REGION Network 80: Check for Parameter Format Type
   RUNG wire#powerrail
      Contact( #ALLWAYS_ON )
      { S7_GenerateENO := "TRUE" } Move(in := #PARA_INTERNAL_DPV1.Responce.Format, out1 => #Response_Format_Dummy)
      wire#w1
      { S7_Templates := "SrcType := Int" } EQ_Contact(in1 := #Response_Format_Dummy, in2 := 67)
      wire#w2
      Coil( #Format_Check_1 )
   END_RUNG
   RUNG wire#w1
      { S7_Templates := "SrcType := Int" } EQ_Contact(in1 := #Response_Format_Dummy, in2 := 4)
   END_RUNG wire#w2
   RUNG wire#w1
      { S7_Templates := "SrcType := Int" } EQ_Contact(in1 := #Response_Format_Dummy, in2 := 7)
   END_RUNG wire#w2
   // the same network as SCL:
   // ENO of a box is taken as its EN; it also drops when the box reports an error
   IF #ALLWAYS_ON THEN #Response_Format_Dummy := #PARA_INTERNAL_DPV1.Responce.Format; END_IF;
   #Format_Check_1 := #ALLWAYS_ON AND ((#Response_Format_Dummy = 67) OR (#Response_Format_Dummy = 4) OR (#Response_Format_Dummy = 7));
END_REGION

REGION Network 81: Wrtie parameter area DP-V1
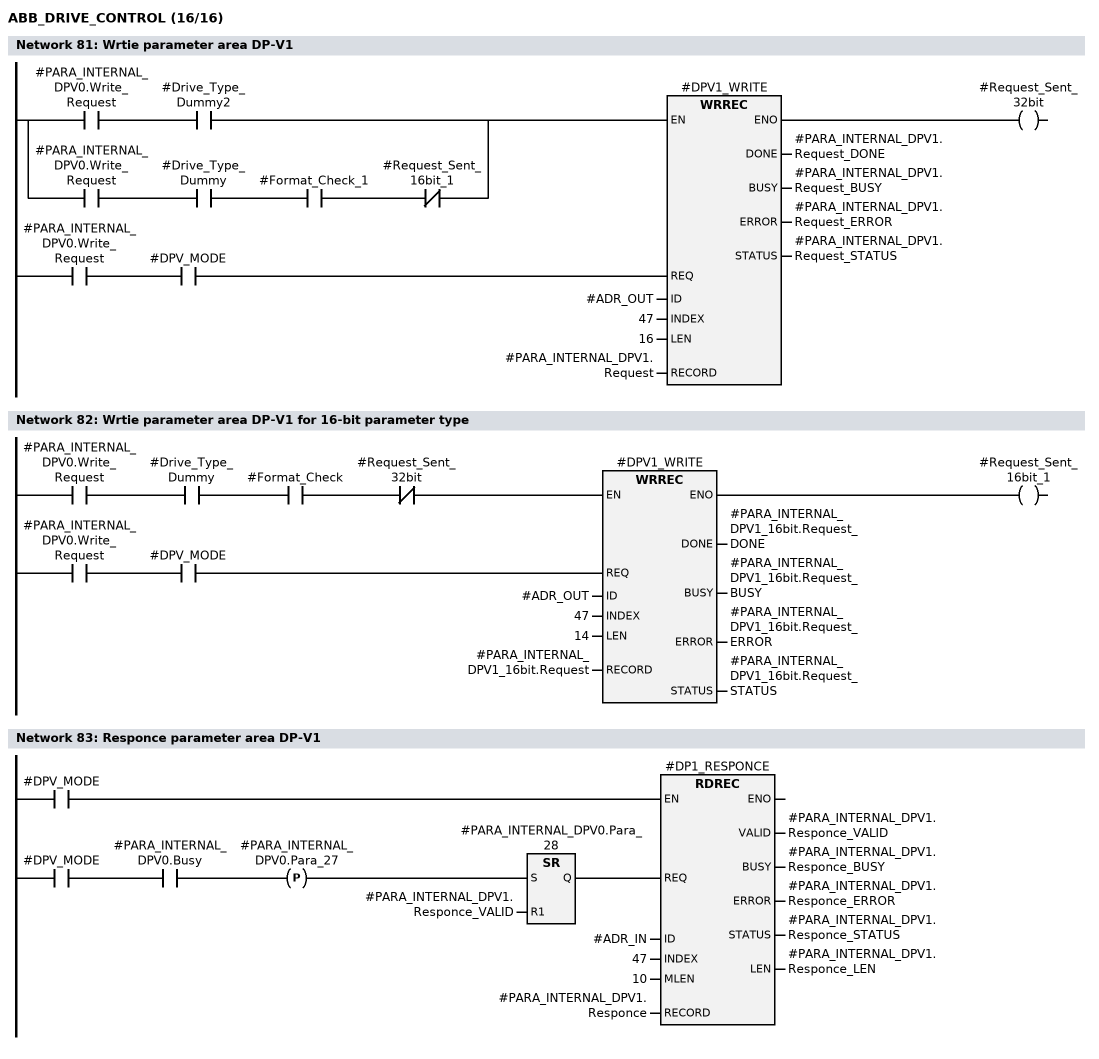
   // ENO of a box is taken as its EN; it also drops when the box reports an error
   #_w1 := (#PARA_INTERNAL_DPV0.Write_Request AND #Drive_Type_Dummy2) OR (#PARA_INTERNAL_DPV0.Write_Request AND #Drive_Type_Dummy AND #Format_Check_1 AND NOT #Request_Sent_16bit_1);
   IF #_w1 THEN
       #DPV1_WRITE(REQ := #PARA_INTERNAL_DPV0.Write_Request AND #DPV_MODE,   // WRREC
                   ID := #ADR_OUT,
                   INDEX := 47,
                   LEN := 16,
                   RECORD := #PARA_INTERNAL_DPV1.Request,
                   DONE => #PARA_INTERNAL_DPV1.Request_DONE,
                   BUSY => #PARA_INTERNAL_DPV1.Request_BUSY,
                   ERROR => #PARA_INTERNAL_DPV1.Request_ERROR,
                   STATUS => #PARA_INTERNAL_DPV1.Request_STATUS);
   END_IF;
   #Request_Sent_32bit := #_w1;
END_REGION

REGION Network 82: Wrtie parameter area DP-V1 for 16-bit parameter type
   // ENO of a box is taken as its EN; it also drops when the box reports an error
   #_w1 := #PARA_INTERNAL_DPV0.Write_Request AND #Drive_Type_Dummy AND #Format_Check AND NOT #Request_Sent_32bit;
   IF #_w1 THEN
       #DPV1_WRITE(REQ := #PARA_INTERNAL_DPV0.Write_Request AND #DPV_MODE,   // WRREC
                   ID := #ADR_OUT,
                   INDEX := 47,
                   LEN := 14,
                   RECORD := #PARA_INTERNAL_DPV1_16bit.Request,
                   DONE => #PARA_INTERNAL_DPV1_16bit.Request_DONE,
                   BUSY => #PARA_INTERNAL_DPV1_16bit.Request_BUSY,
                   ERROR => #PARA_INTERNAL_DPV1_16bit.Request_ERROR,
                   STATUS => #PARA_INTERNAL_DPV1_16bit.Request_STATUS);
   END_IF;
   #Request_Sent_16bit_1 := #_w1;
END_REGION

REGION Network 83: Responce parameter area DP-V1
   #_w1 := #DPV_MODE AND #PARA_INTERNAL_DPV0.Busy;
   #_w2 := #_w1 AND NOT #PARA_INTERNAL_DPV0.Para_27;   // rising edge
   #PARA_INTERNAL_DPV0.Para_27 := #_w1;
   IF #_w2 THEN
       #PARA_INTERNAL_DPV0.Para_28 := TRUE;   // SR flip-flop
   END_IF;
   IF #PARA_INTERNAL_DPV1.Responce_VALID THEN #PARA_INTERNAL_DPV0.Para_28 := FALSE; END_IF;
   IF #DPV_MODE THEN
       #DP1_RESPONCE(REQ := #PARA_INTERNAL_DPV0.Para_28,   // RDREC
                     ID := #ADR_IN,
                     INDEX := 47,
                     MLEN := 10,
                     RECORD := #PARA_INTERNAL_DPV1.Responce,
                     VALID => #PARA_INTERNAL_DPV1.Responce_VALID,
                     BUSY => #PARA_INTERNAL_DPV1.Responce_BUSY,
                     ERROR => #PARA_INTERNAL_DPV1.Responce_ERROR,
                     STATUS => #PARA_INTERNAL_DPV1.Responce_STATUS,
                     LEN => #PARA_INTERNAL_DPV1.Responce_LEN);
   END_IF;
END_REGION
END_FUNCTION_BLOCK

FUNCTION_BLOCK "ACS_DRIVE_PARA"   // FB501, LAD
TITLE = ACS_DRIVE_PARA
{ S7_Optimized_Access := 'FALSE' }
AUTHOR : ABB
FAMILY : DRIVES
NAME : ABB
VERSION : 1.2
   VAR_INPUT
      ADR_IN : Hw_Io;   // 1: Address of first input byte
      ADR_OUT : Hw_Io;   // 2: Address of first output byte
      READ : Bool;   // 3: Read parameter value
      WRITE : Bool;   // 4: Write parameter value
      PARAM_NUM : DInt;   // 5: Parameter number: 3 digits = group, 2 digits = index; e.g Par 20.06 = 2006
      VALUE_IN : DInt;   // 6: Write parameter value
      DRIVE : DB_ANY;   // 8: Instance of the ABB_DRIVE_CONTROL_FB
      THIS_BLOCK_DB : DB_ANY;
   END_VAR
   VAR_OUTPUT
      DONE : Bool;   // 1: Pulse execution finished
      ERR : Bool;   // 2: Error occured
      ERNO : Word;   // 3: Error ID
      BUSY : Bool;   // 4: Function block busy
      PARAM_NUM_OUT : DInt;   // 5: Parameter number: 3 digits = group, 2 digits = index; e.g Par 20.06 = 2006
      VALUE_OUT : DInt;   // 6: Readed parameter value
   END_VAR
   VAR
      PARA_INTERNAL : Struct
         Done : Bool;
         Err : Bool;
         Busy : Bool;
         Read_FB : Bool;
         Write_FB : Bool;
         Time_out : Bool;
         Read_request : Bool;
         Write_Request : Bool;
         Parameter_access : Bool;
         para_err : Bool;
         Para_10 : Bool;
         DPV1_DONE : Bool;
         Para_12 : Bool;
         Para_13 : Bool;
         Para_14 : Bool;
         Para_15 : Bool;
         Para_16 : Bool;
         Para_17 : Bool;
         Para_18 : Bool;
         Para_19 : Bool;
         Para_20 : Bool;
         Para_21 : Bool;
         Para_22 : Bool;
         Para_23 : Bool;
         Para_24 : Bool;
         Para_25 : Bool;
         Para_26 : Bool;
         Para_27 : Bool;
         Para_28 : Bool;
         Para_29 : Bool;
         Para_30 : Bool;
         DPV_MODE : Bool;   // DP-V0 = 0 (false) / DP-V1 = 1 (true)
         RESPONCE_LABEL : Int;
         PARA_NUM_OUT : Int;
         PARA_NUM_INDEX_OUT : Int;
         PARA_ERR_NRO : Word;
         PARA_VALUE_OUT : DInt;
         ADDRESS_IN : Word;
         ADDRESS_OUT : Word;
         Master_to_Slave : Struct
            ID : Word;   // Request Label bits 4-7 Parameter number bits 0-2
            IND : Word;   // Parameter number index bits 0-15
            VALUE : DWord;   // Parameter values
         END_STRUCT;
         Slave_to_Master : Struct
            ID : Word;   // Request Label bits 4-7 Parameter number bits 0-2
            IND : Word;   // Parameter number index bits 0-15
            VALUE : DWord;   // Parameter values
         END_STRUCT;
         PPO_TYPE : Int;   // PPO-Type: 1,2,3,4,5 or 6; 0 = no function
         ADAPTER_TYPE : Int;   // AdapterType:FPBA=1,RPBA=2,FENA=3
         DRIVE_TYPE : Int;   // ACS800=1,ACSM1=2,ACS350=3,ACS355=4,ACS550=5,ACS850=6,ACS880=7,ACS580=8,ACS380=9
      END_STRUCT;
      ReadCommand : Int;
      WriteCommand : Int;
      PARA_NUM_IN : Int;
      PARA_NUM_ON_RPBA : Bool;
      PARA_NUM_ON_FPBA : Bool;
      PARANUM_DINT : DInt;
      PARA_ERR : Bool;
      ITERNAL_READ_ERR : Int;
      ITERNAL_ERITE_ERR : Int;
      TEMP_PARA_NUM : DInt;
      Allways_ON : Bool;
      Allways_OFF : Bool;
      Dummy : Bool;
      TEMPPI : DInt;
      START_VALUE : DInt;
      ZERO_VALUE : DInt;
      PARA_INTERNAL_DPV1 : Struct
         Request : Struct
            Reference : Byte;
            ID : Byte;
            Axis : Byte;
            NoOfParameters : Byte;
            Attribute : Byte;
            NoOfElements : Byte;
            ParameterIndex : Word;
            Subindex : Word;
            Format : Byte;
            NumberOfValues : Byte;
            Value : DWord;
         END_STRUCT;
         Responce : Struct
            Reference : Byte;
            ID : Byte;
            Axis : Byte;
            NoOfParametrs : Byte;
            Format : Byte;
            NoOfValues : Byte;
            Value : DWord;
         END_STRUCT;
         Request_DONE : Bool;
         Request_BUSY : Bool;
         Request_ERROR : Bool;
         Request_STATUS : DWord;
         Responce_VALID : Bool;
         Responce_BUSY : Bool;
         Responce_ERROR : Bool;
         Responce_STATUS : DWord;
         Responce_LEN : UInt;
      END_STRUCT;
      Drive_Dummy1 : Bool;
      Drive_Dummy2 : Bool;
      PARA_INTERNAL_DPV1_16bit : Struct
         Request : Struct
            Reference : Byte;
            ID : Byte;
            Axis : Byte;
            NoOfParameters : Byte;
            Attribute : Byte;
            NoOfElements : Byte;
            ParameterIndex : Word;
            Subindex : Word;
            Format : Byte;
            NumberOfValues : Byte;
            Value : Word;
         END_STRUCT;
         Responce : Struct
            Reference : Byte;
            ID : Byte;
            Axis : Byte;
            NoOfParametrs : Byte;
            Format : Byte;
            NoOfValues : Byte;
            Value : DWord;
         END_STRUCT;
         Request_DONE : Bool;
         Request_BUSY : Bool;
         Request_ERROR : Bool;
         Request_STATUS : DWord;
         Responce_VALID : Bool;
         Responce_BUSY : Bool;
         Responce_ERROR : Bool;
         Responce_STATUS : DWord;
         Responce_LEN : Int;
      END_STRUCT;
      PARA32bit_Read : Bool;
      PARA16bit_Read : Bool;
   END_VAR
   VAR_TEMP
      PARAM_NUM_Temp : Int;
      ReadCommand_Temp : Int;
      PARAM_NUM_Temp2 : Int;
      WriteCommand_Temp : Int;
      PARA_INTERNAL_Slave_to_Master_ID_Temp : Word;
      PARA_INTERNAL_Slave_to_Master_ID_Temp2 : Word;
      PARA_INTERNAL_Slave_to_Master_ID_Temp3 : Word;
      PARA_INTERNAL_Slave_to_Master_IND_Temp : Word;
      PARA_INTERNAL_Master_to_Slave_ID_Temp : DInt;
      PARA_INTERNAL_Master_to_Slave_ID_Num_Temp : DInt;
      PARA_INTERNAL_Master_to_Slave_ID_Num_Temp2 : Int;
      ReadCommand_Temp2 : Word;
      PARA_INTERNAL_Master_to_Slave_ID_Temp2 : DInt;
      PARA_INTERNAL_Master_to_Slave_ID_Num_Temp3 : DInt;
      PARA_INTERNAL_Master_to_Slave_ID_Num_Temp4 : Int;
      WriteCommand_Temp2 : Word;
      PARA_INTERNAL_Slave_to_Master_ID_Temp4 : Word;
      PARA_INTERNAL_Slave_to_Master_ID_Temp5 : Word;
      PARA_INTERNAL_Slave_to_Master_ID_Temp6 : Word;
      PARA_INTERNAL_Slave_to_Master_IND_Temp2 : Word;
      PARA_INTERNAL_DPV1_Request_ParameterIndex_Temp : DInt;
      PARA_INTERNAL_DPV1_Request_ParameterIndex_Temp2 : DInt;
      PARAM_NUM_Temp3 : Int;
      PARAM_NUM_Temp4 : Word;
      PARA_INTERNAL_Slave_to_Master_ID_IND_Temp : DInt;
      PARA_INTERNAL_Slave_to_Master_ID_IND_Temp2 : DInt;
      Dummy_Real : DWord;
      PARA_INTERNAL_DPV1_Responce_Value_Converted : DInt;
      PARA_INTERNAL_ADAPTER_TYPE_Temp : Int;
      VALUE_IN_Conv : Int;
      Error_Return : Int;
   END_VAR
   VAR_TEMP   // added for the SCL form of the ladder/FBD networks
      _w1 : Bool;
      _w2 : Bool;
      _w3 : Bool;
      _w4 : Bool;
   END_VAR
BEGIN

REGION Network 1: Help flags
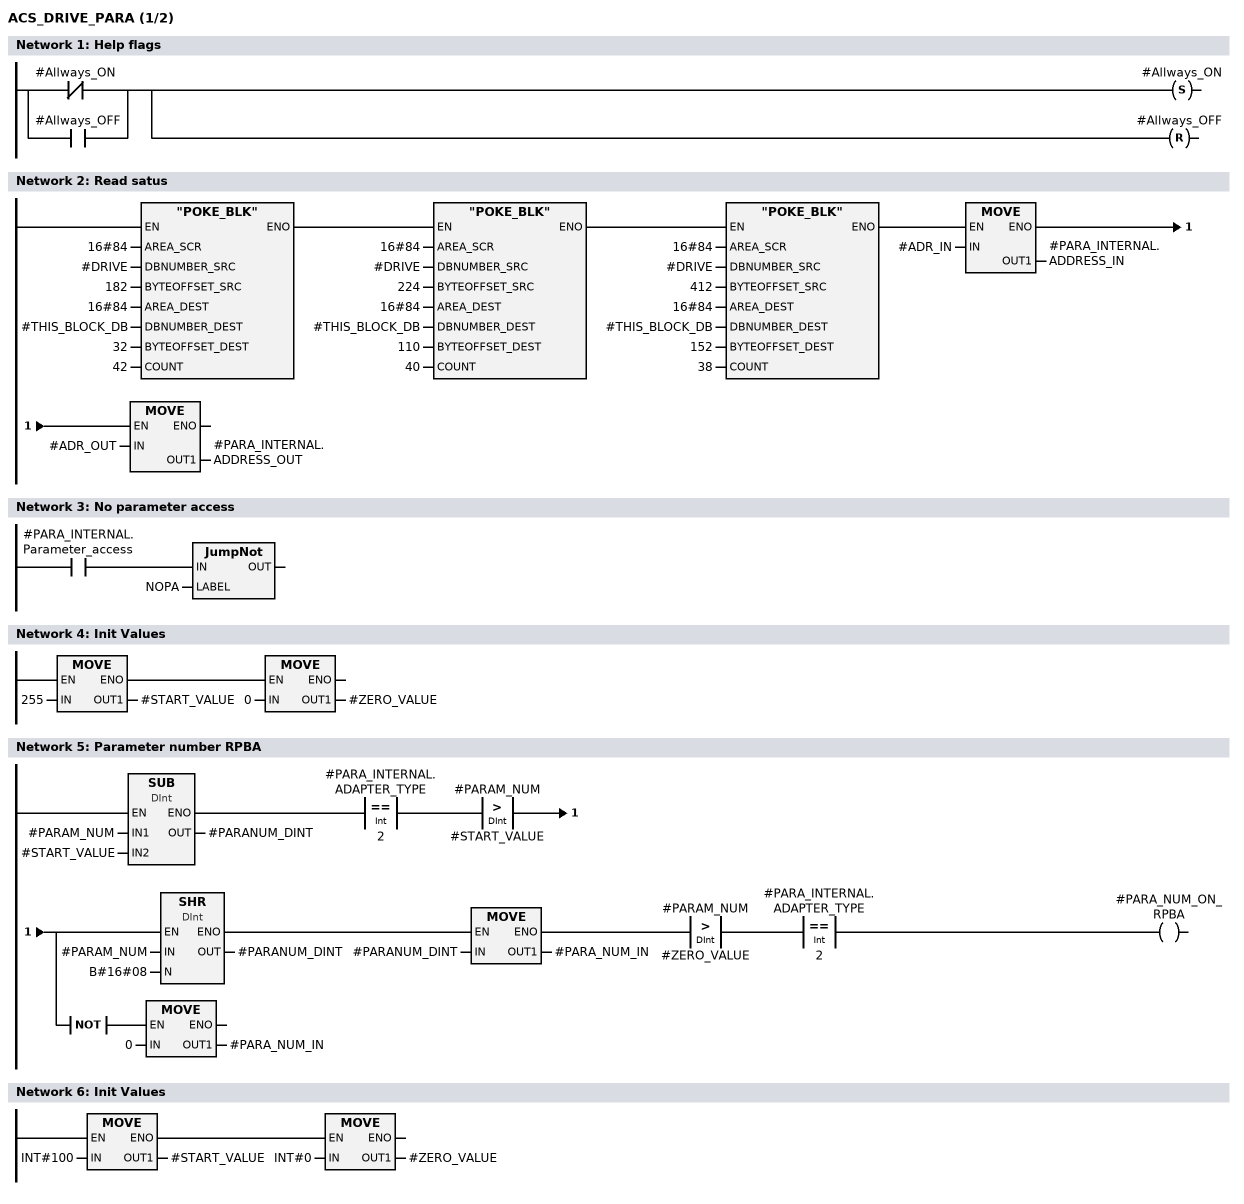
   RUNG wire#powerrail
      I_Contact( #Allways_ON )
      wire#w1
      S_Coil( #Allways_ON )
   END_RUNG
   RUNG wire#powerrail
      Contact( #Allways_OFF )
   END_RUNG wire#w1
   RUNG wire#w1
      R_Coil( #Allways_OFF )
   END_RUNG
   // the same network as SCL:
   #_w1 := NOT #Allways_ON OR #Allways_OFF;
   IF #_w1 THEN
       #Allways_ON := TRUE;
       #Allways_OFF := FALSE;
   END_IF;
END_REGION

REGION Network 2: Read satus
   RUNG wire#powerrail
      "POKE_BLK"(AREA_SCR := 16#84, DBNUMBER_SRC := #DRIVE, BYTEOFFSET_SRC := 182, AREA_DEST := 16#84, DBNUMBER_DEST := #THIS_BLOCK_DB, BYTEOFFSET_DEST := 32, COUNT := 42)
      "POKE_BLK"(AREA_SCR := 16#84, DBNUMBER_SRC := #DRIVE, BYTEOFFSET_SRC := 224, AREA_DEST := 16#84, DBNUMBER_DEST := #THIS_BLOCK_DB, BYTEOFFSET_DEST := 110, COUNT := 40)
      "POKE_BLK"(AREA_SCR := 16#84, DBNUMBER_SRC := #DRIVE, BYTEOFFSET_SRC := 412, AREA_DEST := 16#84, DBNUMBER_DEST := #THIS_BLOCK_DB, BYTEOFFSET_DEST := 152, COUNT := 38)
      { S7_GenerateENO := "TRUE" } Move(in := #ADR_IN, out1 => #PARA_INTERNAL.ADDRESS_IN)
      { S7_GenerateENO := "TRUE" } Move(in := #ADR_OUT, out1 => #PARA_INTERNAL.ADDRESS_OUT)
   END_RUNG
   // the same network as SCL:
   // ENO of a box is taken as its EN; it also drops when the box reports an error
   "POKE_BLK"(AREA_SCR := 16#84,
              DBNUMBER_SRC := #DRIVE,
              BYTEOFFSET_SRC := 182,
              AREA_DEST := 16#84,
              DBNUMBER_DEST := #THIS_BLOCK_DB,
              BYTEOFFSET_DEST := 32,
              COUNT := 42,
              ENO => #_w1);
   "POKE_BLK"(EN := #_w1,
              AREA_SCR := 16#84,
              DBNUMBER_SRC := #DRIVE,
              BYTEOFFSET_SRC := 224,
              AREA_DEST := 16#84,
              DBNUMBER_DEST := #THIS_BLOCK_DB,
              BYTEOFFSET_DEST := 110,
              COUNT := 40,
              ENO => #_w2);
   "POKE_BLK"(EN := #_w2,
              AREA_SCR := 16#84,
              DBNUMBER_SRC := #DRIVE,
              BYTEOFFSET_SRC := 412,
              AREA_DEST := 16#84,
              DBNUMBER_DEST := #THIS_BLOCK_DB,
              BYTEOFFSET_DEST := 152,
              COUNT := 38,
              ENO => #_w3);
   IF #_w3 THEN
       #PARA_INTERNAL.ADDRESS_IN := #ADR_IN;
       #PARA_INTERNAL.ADDRESS_OUT := #ADR_OUT;
   END_IF;
END_REGION

REGION Network 3: No parameter access
   // no SCL statement known for JumpNot: written as a call
   JumpNot(in := #PARA_INTERNAL.Parameter_access, label := NOPA);
END_REGION

REGION Network 4: Init Values
   RUNG wire#powerrail
      { S7_GenerateENO := "TRUE" } Move(in := 255, out1 => #START_VALUE)
      { S7_GenerateENO := "TRUE" } Move(in := 0, out1 => #ZERO_VALUE)
   END_RUNG
   // the same network as SCL:
   // ENO of a box is taken as its EN; it also drops when the box reports an error
   #START_VALUE := 255;
   #ZERO_VALUE := 0;
END_REGION

REGION Network 5: Parameter number RPBA
   RUNG wire#powerrail
      { S7_Templates := "SrcType := DInt"; S7_GenerateENO := "TRUE" } Sub(in1 := #PARAM_NUM, in2 := #START_VALUE, out => #PARANUM_DINT)
      { S7_Templates := "SrcType := Int" } EQ_Contact(in1 := #PARA_INTERNAL.ADAPTER_TYPE, in2 := 2)
      { S7_Templates := "SrcType := DInt" } GT_Contact(in1 := #PARAM_NUM, in2 := #START_VALUE)
      wire#w1
      { S7_Templates := "SrcType := DInt"; S7_GenerateENO := "TRUE" } Shr(in := #PARAM_NUM, n := B#16#08, out => #PARANUM_DINT)
      { S7_GenerateENO := "TRUE" } Move(in := #PARANUM_DINT, out1 => #PARA_NUM_IN)
      { S7_Templates := "SrcType := DInt" } GT_Contact(in1 := #PARAM_NUM, in2 := #ZERO_VALUE)
      { S7_Templates := "SrcType := Int" } EQ_Contact(in1 := #PARA_INTERNAL.ADAPTER_TYPE, in2 := 2)
      Coil( #PARA_NUM_ON_RPBA )
   END_RUNG
   RUNG wire#w1
      Not()
      { S7_GenerateENO := "TRUE" } Move(in := 0, out1 => #PARA_NUM_IN)
   END_RUNG
   // the same network as SCL:
   // ENO of a box is taken as its EN; it also drops when the box reports an error
   #PARANUM_DINT := #PARAM_NUM - #START_VALUE;
   #_w1 := (#PARA_INTERNAL.ADAPTER_TYPE = 2) AND (#PARAM_NUM > #START_VALUE);
   IF #_w1 THEN
       #PARANUM_DINT := SHR(IN := #PARAM_NUM, N := B#16#08);
       #PARA_NUM_IN := #PARANUM_DINT;
   END_IF;
   #PARA_NUM_ON_RPBA := #_w1 AND (#PARAM_NUM > #ZERO_VALUE) AND (#PARA_INTERNAL.ADAPTER_TYPE = 2);
   IF NOT #_w1 THEN #PARA_NUM_IN := 0; END_IF;
END_REGION

REGION Network 6: Init Values
   RUNG wire#powerrail
      { S7_GenerateENO := "TRUE" } Move(in := INT#100, out1 => #START_VALUE)
      { S7_GenerateENO := "TRUE" } Move(in := INT#0, out1 => #ZERO_VALUE)
   END_RUNG
   // the same network as SCL:
   // ENO of a box is taken as its EN; it also drops when the box reports an error
   #START_VALUE := INT#100;
   #ZERO_VALUE := INT#0;
END_REGION

REGION Network 7: Adapter Type
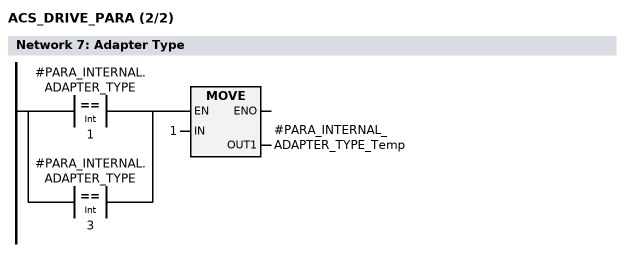
   RUNG wire#powerrail
      { S7_Templates := "SrcType := Int" } EQ_Contact(in1 := #PARA_INTERNAL.ADAPTER_TYPE, in2 := 1)
      wire#w1
      { S7_GenerateENO := "TRUE" } Move(in := 1, out1 => #PARA_INTERNAL_ADAPTER_TYPE_Temp)
   END_RUNG
   RUNG wire#powerrail
      { S7_Templates := "SrcType := Int" } EQ_Contact(in1 := #PARA_INTERNAL.ADAPTER_TYPE, in2 := 3)
   END_RUNG wire#w1
   // the same network as SCL:
   IF (#PARA_INTERNAL.ADAPTER_TYPE = 1) OR (#PARA_INTERNAL.ADAPTER_TYPE = 3) THEN
       #PARA_INTERNAL_ADAPTER_TYPE_Temp := 1;
   END_IF;
END_REGION

REGION Network 8 (FBD): Parameter number FPBA
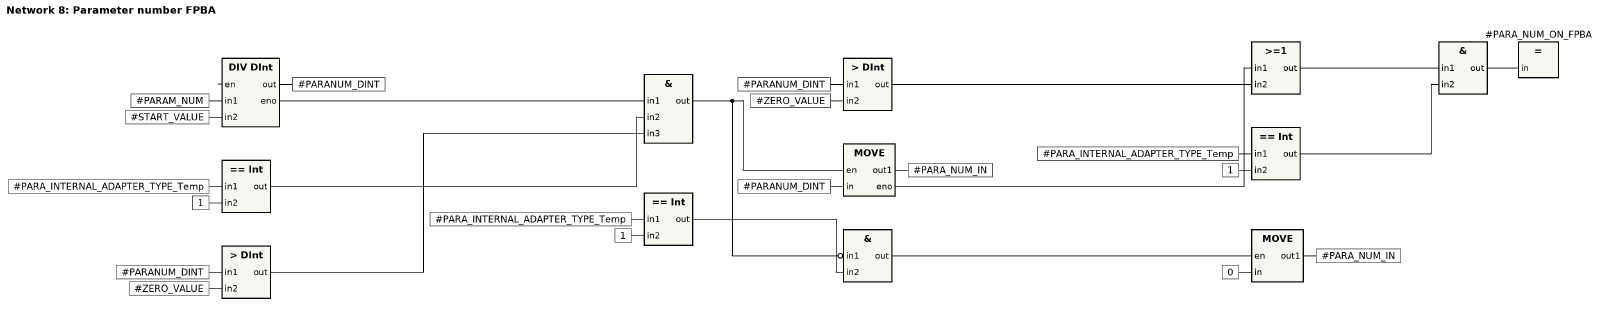
   // ENO of a box is taken as its EN; it also drops when the box reports an error
   #PARANUM_DINT := #PARAM_NUM / #START_VALUE;
   #_w1 := (#PARA_INTERNAL_ADAPTER_TYPE_Temp = 1) AND (#PARANUM_DINT > #ZERO_VALUE);
   IF #_w1 THEN #PARA_NUM_IN := #PARANUM_DINT; END_IF;
   #PARA_NUM_ON_FPBA := (#_w1 OR (#PARANUM_DINT > #ZERO_VALUE)) AND (#PARA_INTERNAL_ADAPTER_TYPE_Temp = 1);
   IF NOT #_w1 AND (#PARA_INTERNAL_ADAPTER_TYPE_Temp = 1) THEN #PARA_NUM_IN := 0; END_IF;
END_REGION

REGION Network 9: Job still active
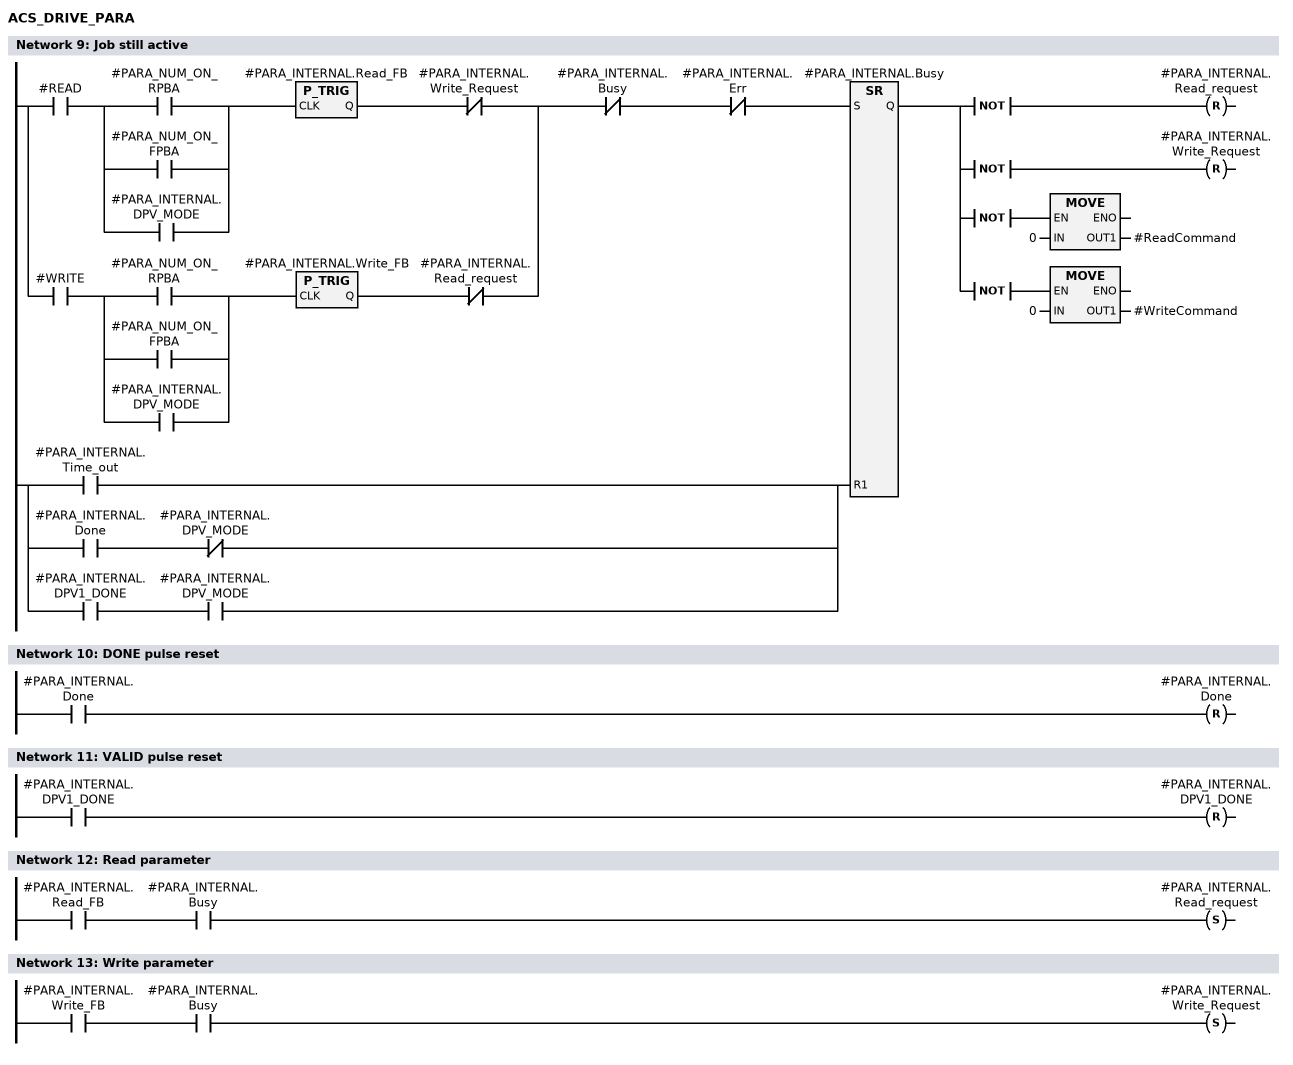
   RUNG wire#powerrail
      Contact( #READ )
      wire#w1
      Contact( #PARA_NUM_ON_RPBA )
      wire#w2
      P_Trig( #PARA_INTERNAL.Read_FB )
      I_Contact( #PARA_INTERNAL.Write_Request )
      wire#w3
      I_Contact( #PARA_INTERNAL.Busy )
      I_Contact( #PARA_INTERNAL.Err )
      S_SR(operand := #PARA_INTERNAL.Busy, r1 := wire#w6)
      wire#w7
      Not()
      R_Coil( #PARA_INTERNAL.Read_request )
   END_RUNG
   RUNG wire#w1
      Contact( #PARA_NUM_ON_FPBA )
   END_RUNG wire#w2
   RUNG wire#w1
      Contact( #PARA_INTERNAL.DPV_MODE )
   END_RUNG wire#w2
   RUNG wire#powerrail
      Contact( #WRITE )
      wire#w4
      Contact( #PARA_NUM_ON_RPBA )
      wire#w5
      P_Trig( #PARA_INTERNAL.Write_FB )
      I_Contact( #PARA_INTERNAL.Read_request )
   END_RUNG wire#w3
   RUNG wire#w4
      Contact( #PARA_NUM_ON_FPBA )
   END_RUNG wire#w5
   RUNG wire#w4
      Contact( #PARA_INTERNAL.DPV_MODE )
   END_RUNG wire#w5
   RUNG wire#powerrail
      Contact( #PARA_INTERNAL.Time_out )
   END_RUNG wire#w6
   RUNG wire#powerrail
      Contact( #PARA_INTERNAL.Done )
      I_Contact( #PARA_INTERNAL.DPV_MODE )
   END_RUNG wire#w6
   RUNG wire#powerrail
      Contact( #PARA_INTERNAL.DPV1_DONE )
      Contact( #PARA_INTERNAL.DPV_MODE )
   END_RUNG wire#w6
   RUNG wire#w7
      Not()
      R_Coil( #PARA_INTERNAL.Write_Request )
   END_RUNG
   RUNG wire#w7
      Not()
      { S7_GenerateENO := "TRUE" } Move(in := 0, out1 => #ReadCommand)
   END_RUNG
   RUNG wire#w7
      Not()
      { S7_GenerateENO := "TRUE" } Move(in := 0, out1 => #WriteCommand)
   END_RUNG
   // the same network as SCL:
   #_w1 := #READ AND (#PARA_NUM_ON_RPBA OR #PARA_NUM_ON_FPBA OR #PARA_INTERNAL.DPV_MODE);
   #_w2 := #_w1 AND NOT #PARA_INTERNAL.Read_FB;   // rising edge
   #PARA_INTERNAL.Read_FB := #_w1;
   #_w3 := #WRITE AND (#PARA_NUM_ON_RPBA OR #PARA_NUM_ON_FPBA OR #PARA_INTERNAL.DPV_MODE);
   #_w4 := #_w3 AND NOT #PARA_INTERNAL.Write_FB;   // rising edge
   #PARA_INTERNAL.Write_FB := #_w3;
   IF ((#_w2 AND NOT #PARA_INTERNAL.Write_Request) OR (#_w4 AND NOT #PARA_INTERNAL.Read_request)) AND NOT #PARA_INTERNAL.Busy AND NOT #PARA_INTERNAL.Err THEN
       #PARA_INTERNAL.Busy := TRUE;   // SR flip-flop
   END_IF;
   IF #PARA_INTERNAL.Time_out OR (#PARA_INTERNAL.Done AND NOT #PARA_INTERNAL.DPV_MODE) OR (#PARA_INTERNAL.DPV1_DONE AND #PARA_INTERNAL.DPV_MODE) THEN
       #PARA_INTERNAL.Busy := FALSE;
   END_IF;
   IF NOT #PARA_INTERNAL.Busy THEN
       #PARA_INTERNAL.Read_request := FALSE;
       #PARA_INTERNAL.Write_Request := FALSE;
       #ReadCommand := 0;
       #WriteCommand := 0;
   END_IF;
END_REGION

REGION Network 10: DONE pulse reset
   RUNG wire#powerrail
      Contact( #PARA_INTERNAL.Done )
      R_Coil( #PARA_INTERNAL.Done )
   END_RUNG
   // the same network as SCL:
   IF #PARA_INTERNAL.Done THEN #PARA_INTERNAL.Done := FALSE; END_IF;
END_REGION

REGION Network 11: VALID pulse reset
   RUNG wire#powerrail
      Contact( #PARA_INTERNAL.DPV1_DONE )
      R_Coil( #PARA_INTERNAL.DPV1_DONE )
   END_RUNG
   // the same network as SCL:
   IF #PARA_INTERNAL.DPV1_DONE THEN #PARA_INTERNAL.DPV1_DONE := FALSE; END_IF;
END_REGION

REGION Network 12: Read parameter
   RUNG wire#powerrail
      Contact( #PARA_INTERNAL.Read_FB )
      Contact( #PARA_INTERNAL.Busy )
      S_Coil( #PARA_INTERNAL.Read_request )
   END_RUNG
   // the same network as SCL:
   IF #PARA_INTERNAL.Read_FB AND #PARA_INTERNAL.Busy THEN #PARA_INTERNAL.Read_request := TRUE; END_IF;
END_REGION

REGION Network 13: Write parameter
   RUNG wire#powerrail
      Contact( #PARA_INTERNAL.Write_FB )
      Contact( #PARA_INTERNAL.Busy )
      S_Coil( #PARA_INTERNAL.Write_Request )
   END_RUNG
   // the same network as SCL:
   IF #PARA_INTERNAL.Write_FB AND #PARA_INTERNAL.Busy THEN #PARA_INTERNAL.Write_Request := TRUE; END_IF;
END_REGION

REGION Network 14 (FBD): Read command
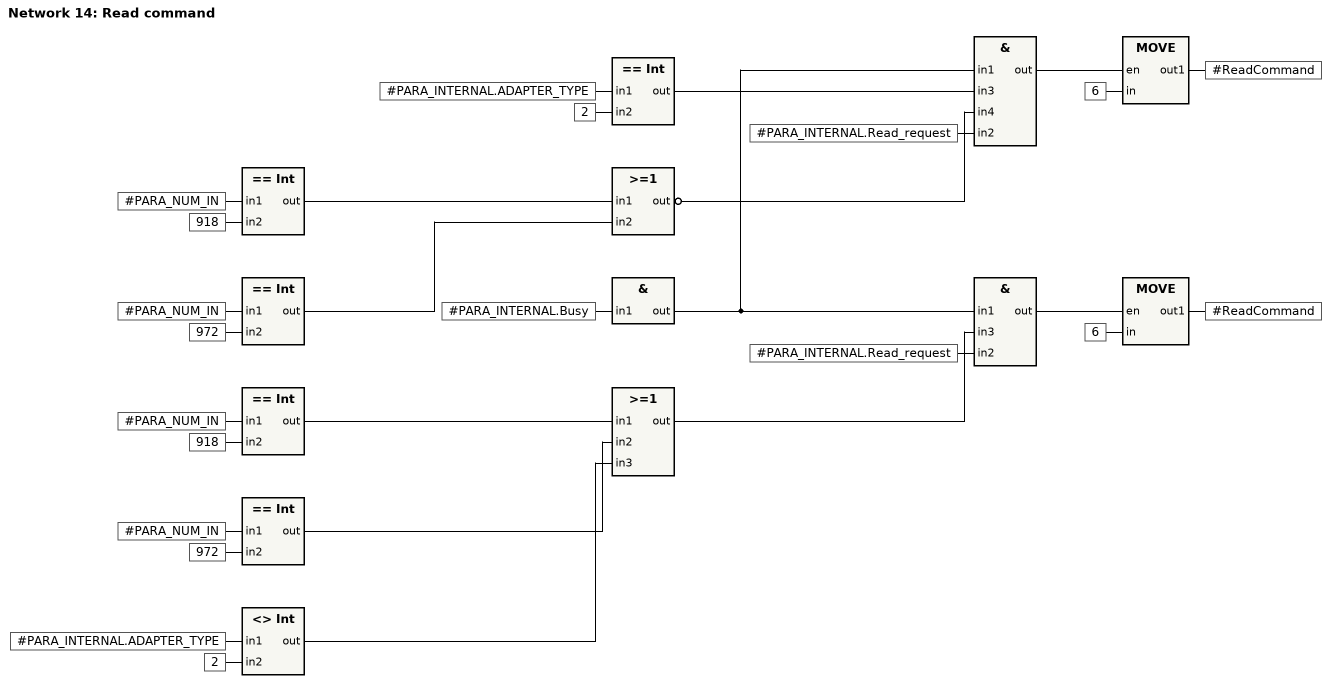
   IF #PARA_INTERNAL.Busy AND (#PARA_INTERNAL.ADAPTER_TYPE = 2) AND NOT ((#PARA_NUM_IN = 918) OR (#PARA_NUM_IN = 972)) AND #PARA_INTERNAL.Read_request THEN
       #ReadCommand := 6;
   END_IF;
   IF #PARA_INTERNAL.Busy AND ((#PARA_NUM_IN = 918) OR (#PARA_NUM_IN = 972) OR (#PARA_INTERNAL.ADAPTER_TYPE <> 2)) AND #PARA_INTERNAL.Read_request THEN
       #ReadCommand := 6;
   END_IF;
END_REGION

REGION Network 15: Write command
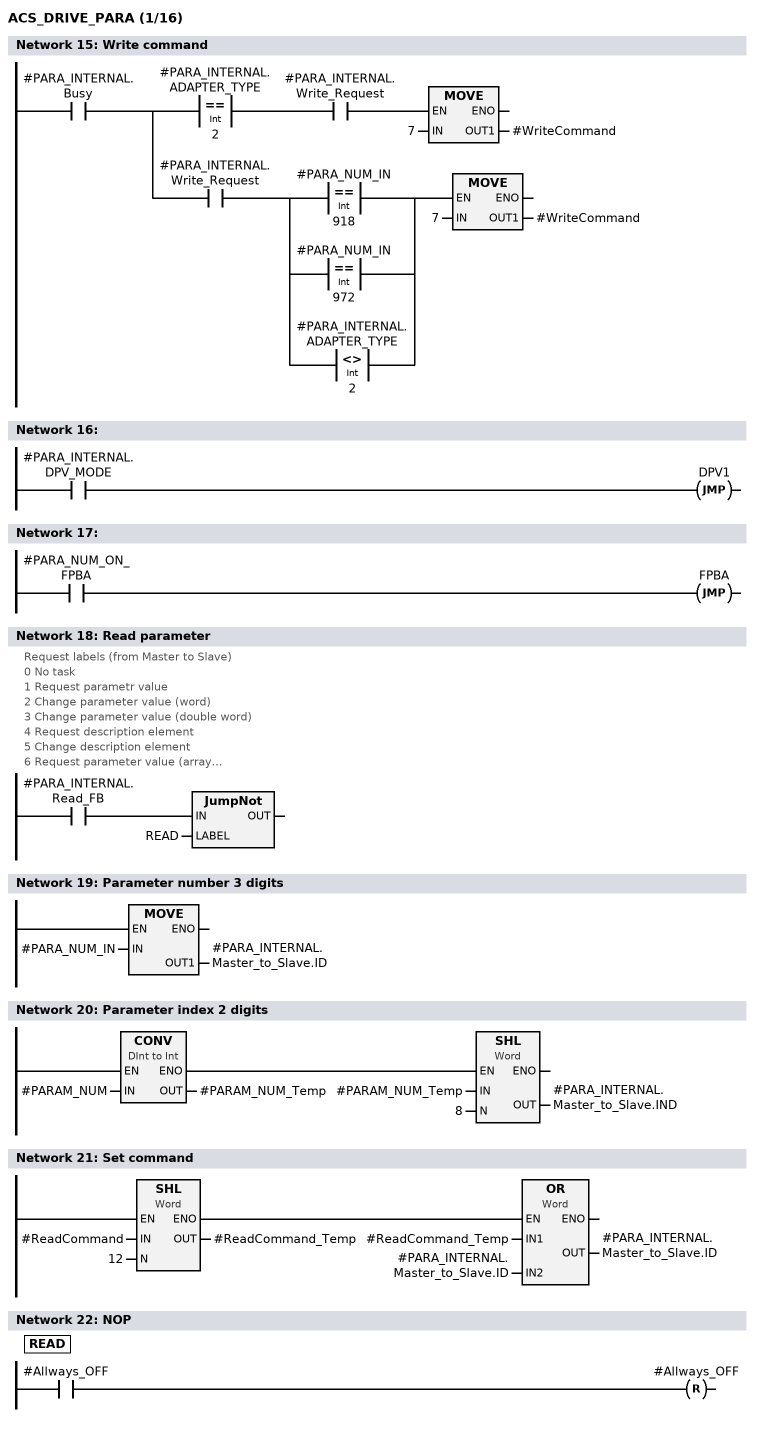
   RUNG wire#powerrail
      Contact( #PARA_INTERNAL.Busy )
      wire#w1
      { S7_Templates := "SrcType := Int" } EQ_Contact(in1 := #PARA_INTERNAL.ADAPTER_TYPE, in2 := 2)
      Contact( #PARA_INTERNAL.Write_Request )
      { S7_GenerateENO := "TRUE" } Move(in := 7, out1 => #WriteCommand)
   END_RUNG
   RUNG wire#w1
      Contact( #PARA_INTERNAL.Write_Request )
      wire#w2
      { S7_Templates := "SrcType := Int" } EQ_Contact(in1 := #PARA_NUM_IN, in2 := 918)
      wire#w3
      { S7_GenerateENO := "TRUE" } Move(in := 7, out1 => #WriteCommand)
   END_RUNG
   RUNG wire#w2
      { S7_Templates := "SrcType := Int" } EQ_Contact(in1 := #PARA_NUM_IN, in2 := 972)
   END_RUNG wire#w3
   RUNG wire#w2
      { S7_Templates := "SrcType := Int" } NE_Contact(in1 := #PARA_INTERNAL.ADAPTER_TYPE, in2 := 2)
   END_RUNG wire#w3
   // the same network as SCL:
   IF #PARA_INTERNAL.Busy AND (#PARA_INTERNAL.ADAPTER_TYPE = 2) AND #PARA_INTERNAL.Write_Request THEN
       #WriteCommand := 7;
   END_IF;
   IF #PARA_INTERNAL.Busy AND #PARA_INTERNAL.Write_Request AND ((#PARA_NUM_IN = 918) OR (#PARA_NUM_IN = 972) OR (#PARA_INTERNAL.ADAPTER_TYPE <> 2)) THEN
       #WriteCommand := 7;
   END_IF;
END_REGION

REGION Network 16
   RUNG wire#powerrail
      Contact( #PARA_INTERNAL.DPV_MODE )
      JumpCoil( DPV1 )
   END_RUNG
   // the same network as SCL:
   IF #PARA_INTERNAL.DPV_MODE THEN GOTO DPV1; END_IF;
END_REGION

REGION Network 17
   RUNG wire#powerrail
      Contact( #PARA_NUM_ON_FPBA )
      JumpCoil( FPBA )
   END_RUNG
   // the same network as SCL:
   IF #PARA_NUM_ON_FPBA THEN GOTO FPBA; END_IF;
END_REGION

REGION Network 18: Read parameter
   // Request labels (from Master to Slave)
   //  0 No task
   // 1 Request parametr value  
   // 2 Change parameter value (word)  
   // 3 Change parameter value (double word)  
   // 4 Request description element  
   // 5 Change description element  
   // 6 Request parameter value (array)  
   // 7 Change parameter value (array word)  
   // 8 Change parameter value (array double word)  
   // 9 Request number of array elements   
   // 
   // Read parameter
   // no SCL statement known for JumpNot: written as a call
   JumpNot(in := #PARA_INTERNAL.Read_FB, label := READ);
END_REGION

REGION Network 19: Parameter number 3 digits
   RUNG wire#powerrail
      { S7_GenerateENO := "TRUE" } Move(in := #PARA_NUM_IN, out1 => #PARA_INTERNAL.Master_to_Slave.ID)
   END_RUNG
   // the same network as SCL:
   #PARA_INTERNAL.Master_to_Slave.ID := #PARA_NUM_IN;
END_REGION

REGION Network 20: Parameter index 2 digits
   RUNG wire#powerrail
      { S7_Templates := "[SrcType := DInt, DestType := Int]"; S7_GenerateENO := "TRUE" } Convert(in := #PARAM_NUM, out => #PARAM_NUM_Temp)
      { S7_Templates := "SrcType := Word"; S7_GenerateENO := "TRUE" } Shl(in := #PARAM_NUM_Temp, n := 8, out => #PARA_INTERNAL.Master_to_Slave.IND)
   END_RUNG
   // the same network as SCL:
   // ENO of a box is taken as its EN; it also drops when the box reports an error
   #PARAM_NUM_Temp := DINT_TO_INT(#PARAM_NUM);
   #PARA_INTERNAL.Master_to_Slave.IND := SHL(IN := #PARAM_NUM_Temp, N := 8);
END_REGION

REGION Network 21: Set command
   // ENO of a box is taken as its EN; it also drops when the box reports an error
   #ReadCommand_Temp := SHL(IN := #ReadCommand, N := 12);
   #PARA_INTERNAL.Master_to_Slave.ID := #ReadCommand_Temp OR #PARA_INTERNAL.Master_to_Slave.ID;
END_REGION

REGION Network 22: NOP
   Label( READ )
   RUNG wire#powerrail
      Contact( #Allways_OFF )
      R_Coil( #Allways_OFF )
   END_RUNG
   // the same network as SCL:
   READ:
   IF #Allways_OFF THEN #Allways_OFF := FALSE; END_IF;
END_REGION

REGION Network 23: Write parameter
   // Request labels (from Master to Slave)
   // 0 No task
   // 1 Request parametr value
   // 2 Change parameter value (word)
   // 3 Change parameter value (double word)
   // 4 Request description element
   // 5 Change description element
   // 6 Request parameter value (array)
   // 7 Change parameter value (array word)
   // 8 Change parameter value (array double word)
   // 9 Request number of array elements
   // 
   //  Write parameter
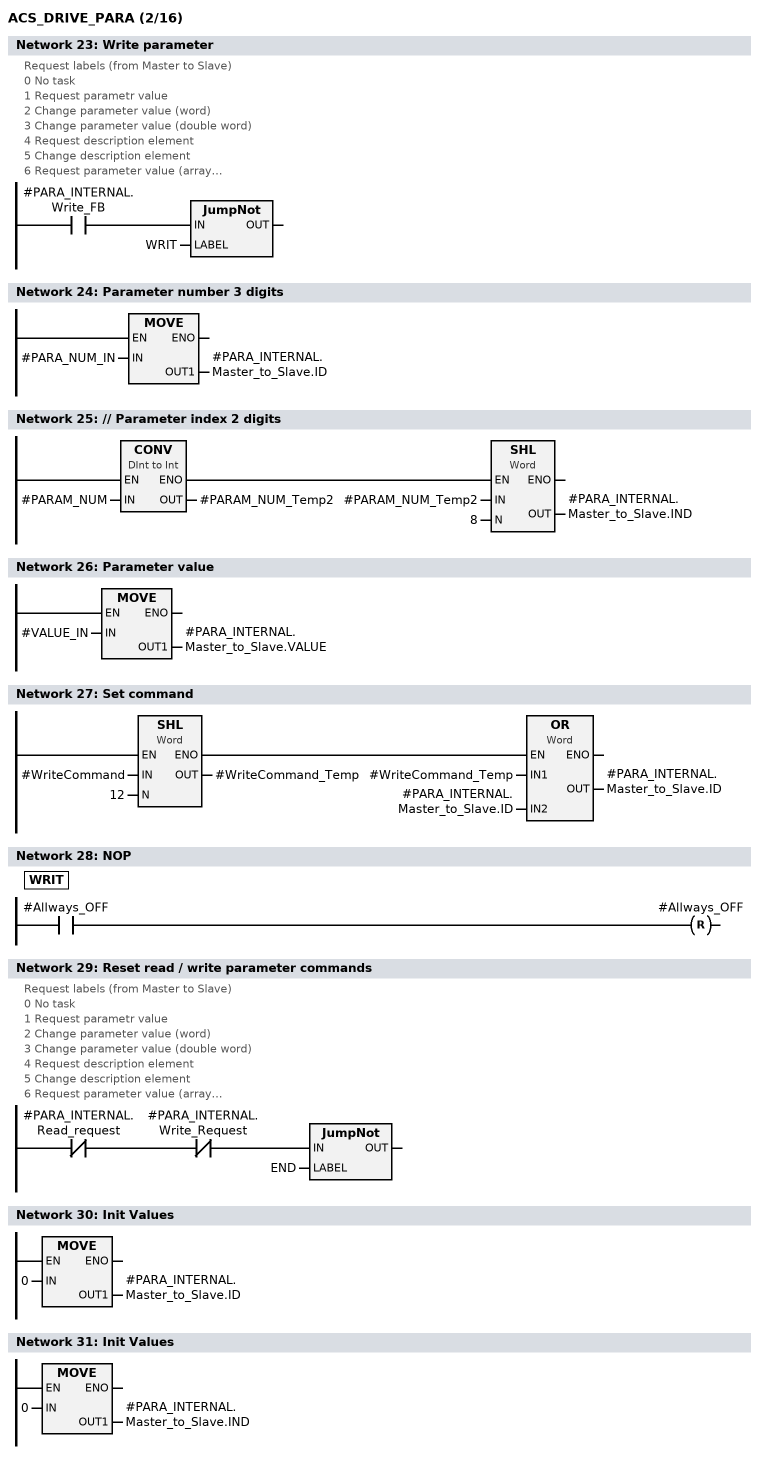
   // no SCL statement known for JumpNot: written as a call
   JumpNot(in := #PARA_INTERNAL.Write_FB, label := WRIT);
END_REGION

REGION Network 24: Parameter number 3 digits
   RUNG wire#powerrail
      { S7_GenerateENO := "TRUE" } Move(in := #PARA_NUM_IN, out1 => #PARA_INTERNAL.Master_to_Slave.ID)
   END_RUNG
   // the same network as SCL:
   #PARA_INTERNAL.Master_to_Slave.ID := #PARA_NUM_IN;
END_REGION

REGION Network 25: // Parameter index 2 digits
   RUNG wire#powerrail
      { S7_Templates := "[SrcType := DInt, DestType := Int]"; S7_GenerateENO := "TRUE" } Convert(in := #PARAM_NUM, out => #PARAM_NUM_Temp2)
      { S7_Templates := "SrcType := Word"; S7_GenerateENO := "TRUE" } Shl(in := #PARAM_NUM_Temp2, n := 8, out => #PARA_INTERNAL.Master_to_Slave.IND)
   END_RUNG
   // the same network as SCL:
   // ENO of a box is taken as its EN; it also drops when the box reports an error
   #PARAM_NUM_Temp2 := DINT_TO_INT(#PARAM_NUM);
   #PARA_INTERNAL.Master_to_Slave.IND := SHL(IN := #PARAM_NUM_Temp2, N := 8);
END_REGION

REGION Network 26: Parameter value
   RUNG wire#powerrail
      { S7_GenerateENO := "TRUE" } Move(in := #VALUE_IN, out1 => #PARA_INTERNAL.Master_to_Slave.VALUE)
   END_RUNG
   // the same network as SCL:
   #PARA_INTERNAL.Master_to_Slave.VALUE := #VALUE_IN;
END_REGION

REGION Network 27: Set command
   // ENO of a box is taken as its EN; it also drops when the box reports an error
   #WriteCommand_Temp := SHL(IN := #WriteCommand, N := 12);
   #PARA_INTERNAL.Master_to_Slave.ID := #WriteCommand_Temp OR #PARA_INTERNAL.Master_to_Slave.ID;
END_REGION

REGION Network 28: NOP
   Label( WRIT )
   RUNG wire#powerrail
      Contact( #Allways_OFF )
      R_Coil( #Allways_OFF )
   END_RUNG
   // the same network as SCL:
   WRIT:
   IF #Allways_OFF THEN #Allways_OFF := FALSE; END_IF;
END_REGION

REGION Network 29: Reset read / write parameter commands
   // Request labels (from Master to Slave)
   // 0 No task
   // 1 Request parametr value
   // 2 Change parameter value (word)
   // 3 Change parameter value (double word)
   // 4 Request description element
   // 5 Change description element
   // 6 Request parameter value (array)
   // 7 Change parameter value (array word)
   // 8 Change parameter value (array double word)
   // 9 Request number of array elements
   // 
   //  Reset parmeter commands
   // no SCL statement known for JumpNot: written as a call
   JumpNot(in := NOT #PARA_INTERNAL.Read_request AND NOT #PARA_INTERNAL.Write_Request, label := END);
END_REGION

REGION Network 30: Init Values
   RUNG wire#powerrail
      { S7_GenerateENO := "TRUE" } Move(in := 0, out1 => #PARA_INTERNAL.Master_to_Slave.ID)
   END_RUNG
   // the same network as SCL:
   #PARA_INTERNAL.Master_to_Slave.ID := 0;
END_REGION

REGION Network 31: Init Values
   RUNG wire#powerrail
      { S7_GenerateENO := "TRUE" } Move(in := 0, out1 => #PARA_INTERNAL.Master_to_Slave.IND)
   END_RUNG
   // the same network as SCL:
   #PARA_INTERNAL.Master_to_Slave.IND := 0;
END_REGION

REGION Network 32: Init Values
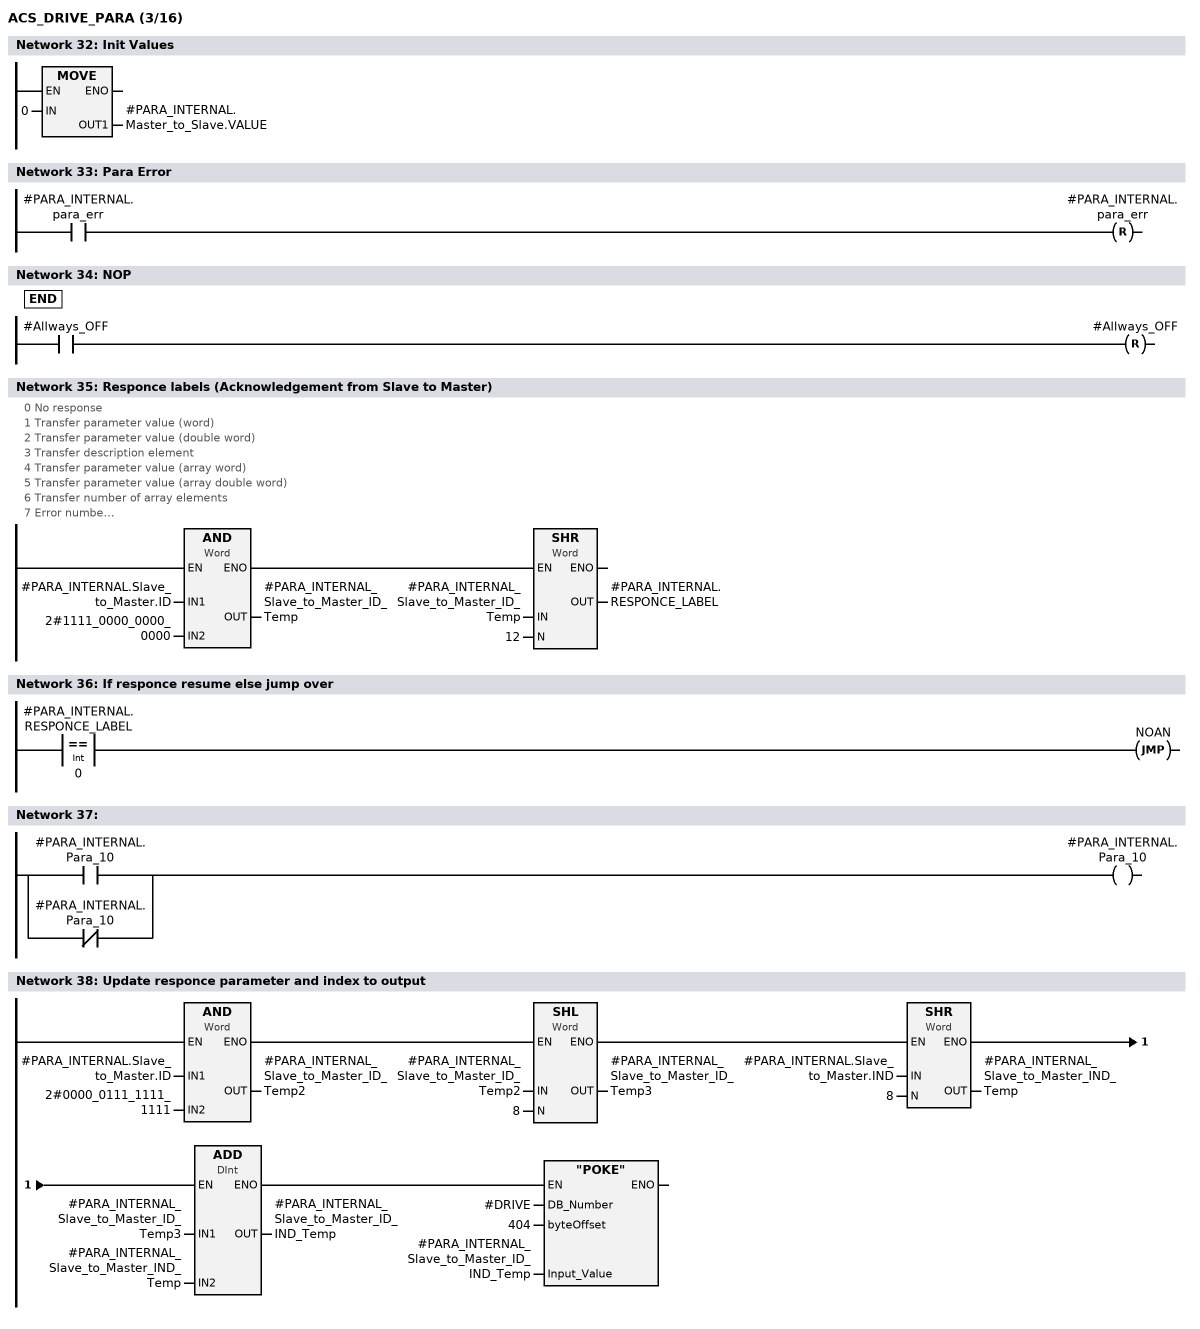
   RUNG wire#powerrail
      { S7_GenerateENO := "TRUE" } Move(in := 0, out1 => #PARA_INTERNAL.Master_to_Slave.VALUE)
   END_RUNG
   // the same network as SCL:
   #PARA_INTERNAL.Master_to_Slave.VALUE := 0;
END_REGION

REGION Network 33: Para Error
   RUNG wire#powerrail
      Contact( #PARA_INTERNAL.para_err )
      R_Coil( #PARA_INTERNAL.para_err )
   END_RUNG
   // the same network as SCL:
   IF #PARA_INTERNAL.para_err THEN #PARA_INTERNAL.para_err := FALSE; END_IF;
END_REGION

REGION Network 34: NOP
   Label( END )
   RUNG wire#powerrail
      Contact( #Allways_OFF )
      R_Coil( #Allways_OFF )
   END_RUNG
   // the same network as SCL:
   END:
   IF #Allways_OFF THEN #Allways_OFF := FALSE; END_IF;
END_REGION

REGION Network 35: Responce labels (Acknowledgement from Slave to Master)
   // 0 No response
   // 1 Transfer parameter value (word)
   // 2 Transfer parameter value (double word)
   // 3 Transfer description element
   // 4 Transfer parameter value (array word)
   // 5 Transfer parameter value (array double word)
   // 6 Transfer number of array elements
   // 7 Error number
   // - 0 Illegal parameter number
   // - 1 Parameter value cannot be changed
   // - 2 Lower or upper limit violated
   // - 3 Error subindex
   // - 4 No array
   // - 5 Incorrect data type
   // - 6 Setting not allowed (can only be reset)
   // - 7 Descriptive element cannot be changed
   // - 9 Descriptive data not available
   // - 11 No parameter change rights
   // - 15 Text array not available
   // - 17 Task cannot be executed due to operating status
   // - 18 Other error
   // - 101 Vendor specific
   // - 102 Request not supported
   // - 103 Request cannot be compeleted due to communication error
   // - 110 Failure during write to non-volatile memory
   // - 111 Request aborted due to time-out
   // - 120 Parameter cannot be mapped to PZD
   // - 121 Parameter cannot be mapped to PZD (end of memory)
   // - 122 Parameter cannot be mapped to PZD (multiple PZD write)
   // - 130 Cannot map Control Word bit (parameter 933-937)
   // - 140 Cannot change mode to TORGUE
   // - 150 Internal buffer overflow
   // - 160 Internal communication error
   // 8 No parameter change rights for PKW interface
   // 9 Parameter data signal (word)
   // 10 Parameter data signal (double word)
   //  Mask responce labels
   RUNG wire#powerrail
      { S7_Templates := "SrcType := Word"; S7_GenerateENO := "TRUE" } And(in1 := #PARA_INTERNAL.Slave_to_Master.ID, in2 := 2#1111_0000_0000_0000, out => #PARA_INTERNAL_Slave_to_Master_ID_Temp)
      { S7_Templates := "SrcType := Word"; S7_GenerateENO := "TRUE" } Shr(in := #PARA_INTERNAL_Slave_to_Master_ID_Temp, n := 12, out => #PARA_INTERNAL.RESPONCE_LABEL)
   END_RUNG
   // the same network as SCL:
   #PARA_INTERNAL_Slave_to_Master_ID_Temp := #PARA_INTERNAL.Slave_to_Master.ID AND 2#1111_0000_0000_0000;
   #PARA_INTERNAL.RESPONCE_LABEL := SHR(IN := #PARA_INTERNAL_Slave_to_Master_ID_Temp, N := 12);
END_REGION

REGION Network 36: If responce resume else jump over
   RUNG wire#powerrail
      { S7_Templates := "SrcType := Int" } EQ_Contact(in1 := #PARA_INTERNAL.RESPONCE_LABEL, in2 := 0)
      JumpCoil( NOAN )
   END_RUNG
   // the same network as SCL:
   IF #PARA_INTERNAL.RESPONCE_LABEL = 0 THEN GOTO NOAN; END_IF;
END_REGION

REGION Network 37
   RUNG wire#powerrail
      Contact( #PARA_INTERNAL.Para_10 )
      wire#w1
      Coil( #PARA_INTERNAL.Para_10 )
   END_RUNG
   RUNG wire#powerrail
      I_Contact( #PARA_INTERNAL.Para_10 )
   END_RUNG wire#w1
   // the same network as SCL:
   #PARA_INTERNAL.Para_10 := #PARA_INTERNAL.Para_10 OR NOT #PARA_INTERNAL.Para_10;
END_REGION

REGION Network 38: Update responce parameter and index to output
   RUNG wire#powerrail
      { S7_Templates := "SrcType := Word"; S7_GenerateENO := "TRUE" } And(in1 := #PARA_INTERNAL.Slave_to_Master.ID, in2 := 2#0000_0111_1111_1111, out => #PARA_INTERNAL_Slave_to_Master_ID_Temp2)
      { S7_Templates := "SrcType := Word"; S7_GenerateENO := "TRUE" } Shl(in := #PARA_INTERNAL_Slave_to_Master_ID_Temp2, n := 8, out => #PARA_INTERNAL_Slave_to_Master_ID_Temp3)
      { S7_Templates := "SrcType := Word"; S7_GenerateENO := "TRUE" } Shr(in := #PARA_INTERNAL.Slave_to_Master.IND, n := 8, out => #PARA_INTERNAL_Slave_to_Master_IND_Temp)
      { S7_Templates := "SrcType := DInt"; S7_GenerateENO := "TRUE" } Add(in1 := #PARA_INTERNAL_Slave_to_Master_ID_Temp3, in2 := #PARA_INTERNAL_Slave_to_Master_IND_Temp, out => #PARA_INTERNAL_Slave_to_Master_ID_IND_Temp)
      "POKE"(DB_Number := #DRIVE, byteOffset := 404, Input_Value := #PARA_INTERNAL_Slave_to_Master_ID_IND_Temp)
   END_RUNG
   // the same network as SCL:
   // ENO of a box is taken as its EN; it also drops when the box reports an error
   #PARA_INTERNAL_Slave_to_Master_ID_Temp2 := #PARA_INTERNAL.Slave_to_Master.ID AND 2#0000_0111_1111_1111;
   #PARA_INTERNAL_Slave_to_Master_ID_Temp3 := SHL(IN := #PARA_INTERNAL_Slave_to_Master_ID_Temp2, N := 8);
   #PARA_INTERNAL_Slave_to_Master_IND_Temp := SHR(IN := #PARA_INTERNAL.Slave_to_Master.IND, N := 8);
   #PARA_INTERNAL_Slave_to_Master_ID_IND_Temp := #PARA_INTERNAL_Slave_to_Master_ID_Temp3 + #PARA_INTERNAL_Slave_to_Master_IND_Temp;
   "POKE"(DB_Number := #DRIVE, byteOffset := 404, Input_Value := #PARA_INTERNAL_Slave_to_Master_ID_IND_Temp);
END_REGION

REGION Network 39: Cheking responce if responce whitout error resume else jump over
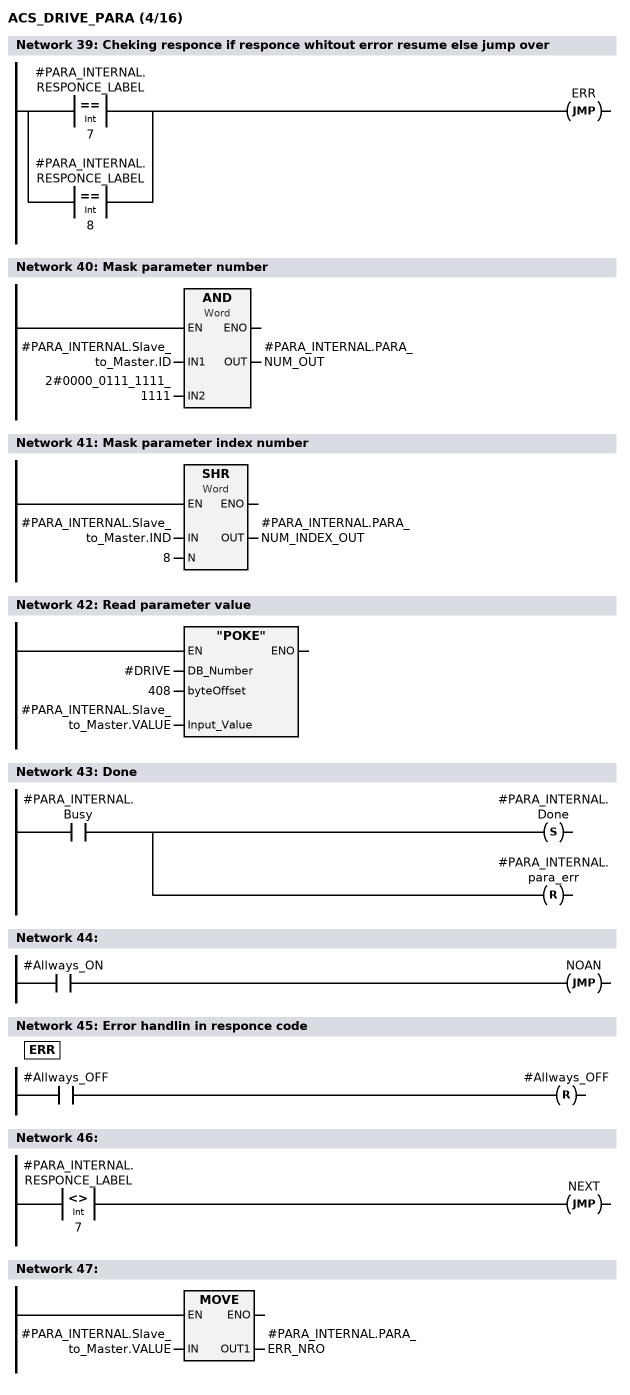
   RUNG wire#powerrail
      { S7_Templates := "SrcType := Int" } EQ_Contact(in1 := #PARA_INTERNAL.RESPONCE_LABEL, in2 := 7)
      wire#w1
      JumpCoil( ERR )
   END_RUNG
   RUNG wire#powerrail
      { S7_Templates := "SrcType := Int" } EQ_Contact(in1 := #PARA_INTERNAL.RESPONCE_LABEL, in2 := 8)
   END_RUNG wire#w1
   // the same network as SCL:
   IF (#PARA_INTERNAL.RESPONCE_LABEL = 7) OR (#PARA_INTERNAL.RESPONCE_LABEL = 8) THEN GOTO ERR; END_IF;
END_REGION

REGION Network 40: Mask parameter number
   RUNG wire#powerrail
      { S7_Templates := "SrcType := Word"; S7_GenerateENO := "TRUE" } And(in1 := #PARA_INTERNAL.Slave_to_Master.ID, in2 := 2#0000_0111_1111_1111, out => #PARA_INTERNAL.PARA_NUM_OUT)
   END_RUNG
   // the same network as SCL:
   #PARA_INTERNAL.PARA_NUM_OUT := #PARA_INTERNAL.Slave_to_Master.ID AND 2#0000_0111_1111_1111;
END_REGION

REGION Network 41: Mask parameter index number
   RUNG wire#powerrail
      { S7_Templates := "SrcType := Word"; S7_GenerateENO := "TRUE" } Shr(in := #PARA_INTERNAL.Slave_to_Master.IND, n := 8, out => #PARA_INTERNAL.PARA_NUM_INDEX_OUT)
   END_RUNG
   // the same network as SCL:
   #PARA_INTERNAL.PARA_NUM_INDEX_OUT := SHR(IN := #PARA_INTERNAL.Slave_to_Master.IND, N := 8);
END_REGION

REGION Network 42: Read parameter value
   RUNG wire#powerrail
      "POKE"(DB_Number := #DRIVE, byteOffset := 408, Input_Value := #PARA_INTERNAL.Slave_to_Master.VALUE)
   END_RUNG
   // the same network as SCL:
   "POKE"(DB_Number := #DRIVE, byteOffset := 408, Input_Value := #PARA_INTERNAL.Slave_to_Master.VALUE);
END_REGION

REGION Network 43: Done
   RUNG wire#powerrail
      Contact( #PARA_INTERNAL.Busy )
      wire#w1
      S_Coil( #PARA_INTERNAL.Done )
   END_RUNG
   RUNG wire#w1
      R_Coil( #PARA_INTERNAL.para_err )
   END_RUNG
   // the same network as SCL:
   IF #PARA_INTERNAL.Busy THEN
       #PARA_INTERNAL.Done := TRUE;
       #PARA_INTERNAL.para_err := FALSE;
   END_IF;
END_REGION

REGION Network 44
   RUNG wire#powerrail
      Contact( #Allways_ON )
      JumpCoil( NOAN )
   END_RUNG
   // the same network as SCL:
   IF #Allways_ON THEN GOTO NOAN; END_IF;
END_REGION

REGION Network 45: Error handlin in responce code
   Label( ERR )
   RUNG wire#powerrail
      Contact( #Allways_OFF )
      R_Coil( #Allways_OFF )
   END_RUNG
   // the same network as SCL:
   ERR:
   IF #Allways_OFF THEN #Allways_OFF := FALSE; END_IF;
END_REGION

REGION Network 46
   RUNG wire#powerrail
      { S7_Templates := "SrcType := Int" } NE_Contact(in1 := #PARA_INTERNAL.RESPONCE_LABEL, in2 := 7)
      JumpCoil( NEXT )
   END_RUNG
   // the same network as SCL:
   IF #PARA_INTERNAL.RESPONCE_LABEL <> 7 THEN GOTO NEXT; END_IF;
END_REGION

REGION Network 47
   RUNG wire#powerrail
      { S7_GenerateENO := "TRUE" } Move(in := #PARA_INTERNAL.Slave_to_Master.VALUE, out1 => #PARA_INTERNAL.PARA_ERR_NRO)
   END_RUNG
   // the same network as SCL:
   #PARA_INTERNAL.PARA_ERR_NRO := #PARA_INTERNAL.Slave_to_Master.VALUE;
END_REGION

REGION Network 48
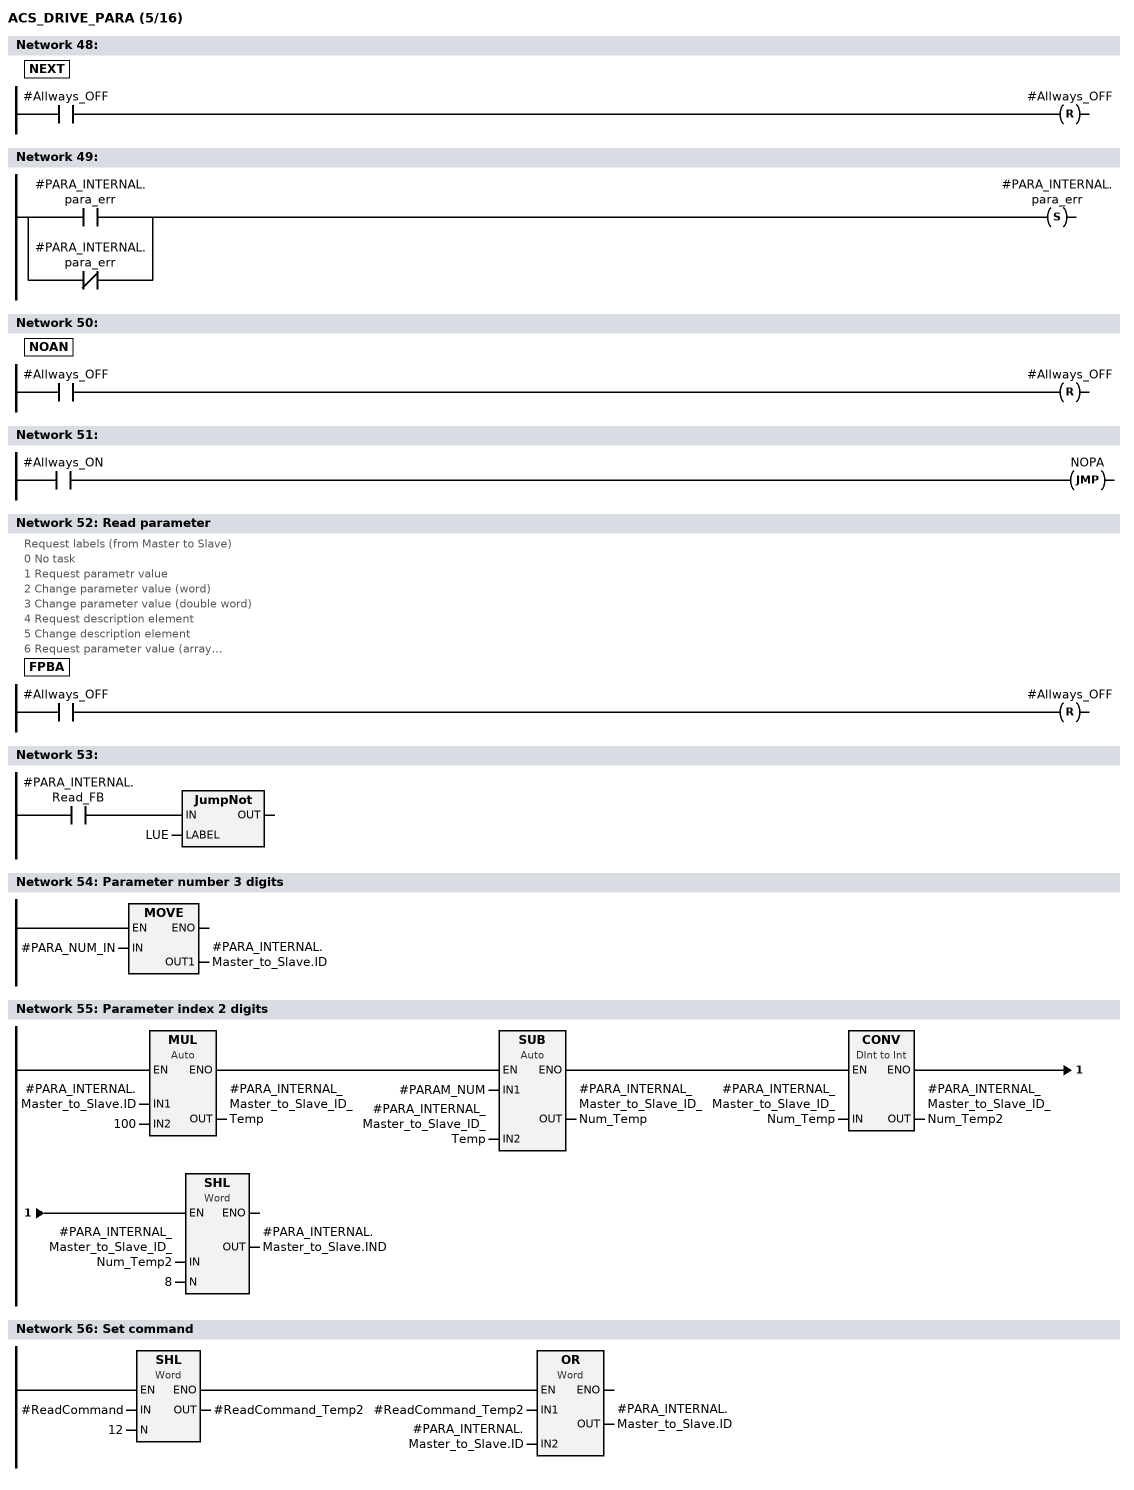
   Label( NEXT )
   RUNG wire#powerrail
      Contact( #Allways_OFF )
      R_Coil( #Allways_OFF )
   END_RUNG
   // the same network as SCL:
   NEXT:
   IF #Allways_OFF THEN #Allways_OFF := FALSE; END_IF;
END_REGION

REGION Network 49
   RUNG wire#powerrail
      Contact( #PARA_INTERNAL.para_err )
      wire#w1
      S_Coil( #PARA_INTERNAL.para_err )
   END_RUNG
   RUNG wire#powerrail
      I_Contact( #PARA_INTERNAL.para_err )
   END_RUNG wire#w1
   // the same network as SCL:
   IF #PARA_INTERNAL.para_err OR NOT #PARA_INTERNAL.para_err THEN #PARA_INTERNAL.para_err := TRUE; END_IF;
END_REGION

REGION Network 50
   Label( NOAN )
   RUNG wire#powerrail
      Contact( #Allways_OFF )
      R_Coil( #Allways_OFF )
   END_RUNG
   // the same network as SCL:
   NOAN:
   IF #Allways_OFF THEN #Allways_OFF := FALSE; END_IF;
END_REGION

REGION Network 51
   RUNG wire#powerrail
      Contact( #Allways_ON )
      JumpCoil( NOPA )
   END_RUNG
   // the same network as SCL:
   IF #Allways_ON THEN GOTO NOPA; END_IF;
END_REGION

REGION Network 52: Read parameter
   // Request labels (from Master to Slave)
   // 0 No task
   // 1 Request parametr value
   // 2 Change parameter value (word)
   // 3 Change parameter value (double word)
   // 4 Request description element
   // 5 Change description element
   // 6 Request parameter value (array)
   // 7 Change parameter value (array word)
   // 8 Change parameter value (array double word)
   // 9 Request number of array elements
   //  Read parameter
   Label( FPBA )
   RUNG wire#powerrail
      Contact( #Allways_OFF )
      R_Coil( #Allways_OFF )
   END_RUNG
   // the same network as SCL:
   FPBA:
   IF #Allways_OFF THEN #Allways_OFF := FALSE; END_IF;
END_REGION

REGION Network 53
   // no SCL statement known for JumpNot: written as a call
   JumpNot(in := #PARA_INTERNAL.Read_FB, label := LUE);
END_REGION

REGION Network 54: Parameter number 3 digits
   RUNG wire#powerrail
      { S7_GenerateENO := "TRUE" } Move(in := #PARA_NUM_IN, out1 => #PARA_INTERNAL.Master_to_Slave.ID)
   END_RUNG
   // the same network as SCL:
   #PARA_INTERNAL.Master_to_Slave.ID := #PARA_NUM_IN;
END_REGION

REGION Network 55: Parameter index 2 digits
   RUNG wire#powerrail
      { S7_GenerateENO := "TRUE" } Mul(in1 := #PARA_INTERNAL.Master_to_Slave.ID, in2 := 100, out => #PARA_INTERNAL_Master_to_Slave_ID_Temp)
      { S7_GenerateENO := "TRUE" } Sub(in1 := #PARAM_NUM, in2 := #PARA_INTERNAL_Master_to_Slave_ID_Temp, out => #PARA_INTERNAL_Master_to_Slave_ID_Num_Temp)
      { S7_Templates := "[SrcType := DInt, DestType := Int]"; S7_GenerateENO := "TRUE" } Convert(in := #PARA_INTERNAL_Master_to_Slave_ID_Num_Temp, out => #PARA_INTERNAL_Master_to_Slave_ID_Num_Temp2)
      { S7_Templates := "SrcType := Word"; S7_GenerateENO := "TRUE" } Shl(in := #PARA_INTERNAL_Master_to_Slave_ID_Num_Temp2, n := 8, out => #PARA_INTERNAL.Master_to_Slave.IND)
   END_RUNG
   // the same network as SCL:
   // ENO of a box is taken as its EN; it also drops when the box reports an error
   #PARA_INTERNAL_Master_to_Slave_ID_Temp := #PARA_INTERNAL.Master_to_Slave.ID * 100;
   #PARA_INTERNAL_Master_to_Slave_ID_Num_Temp := #PARAM_NUM - #PARA_INTERNAL_Master_to_Slave_ID_Temp;
   #PARA_INTERNAL_Master_to_Slave_ID_Num_Temp2 := DINT_TO_INT(#PARA_INTERNAL_Master_to_Slave_ID_Num_Temp);
   #PARA_INTERNAL.Master_to_Slave.IND := SHL(IN := #PARA_INTERNAL_Master_to_Slave_ID_Num_Temp2, N := 8);
END_REGION

REGION Network 56: Set command
   // ENO of a box is taken as its EN; it also drops when the box reports an error
   #ReadCommand_Temp2 := SHL(IN := #ReadCommand, N := 12);
   #PARA_INTERNAL.Master_to_Slave.ID := #ReadCommand_Temp2 OR #PARA_INTERNAL.Master_to_Slave.ID;
END_REGION

REGION Network 57
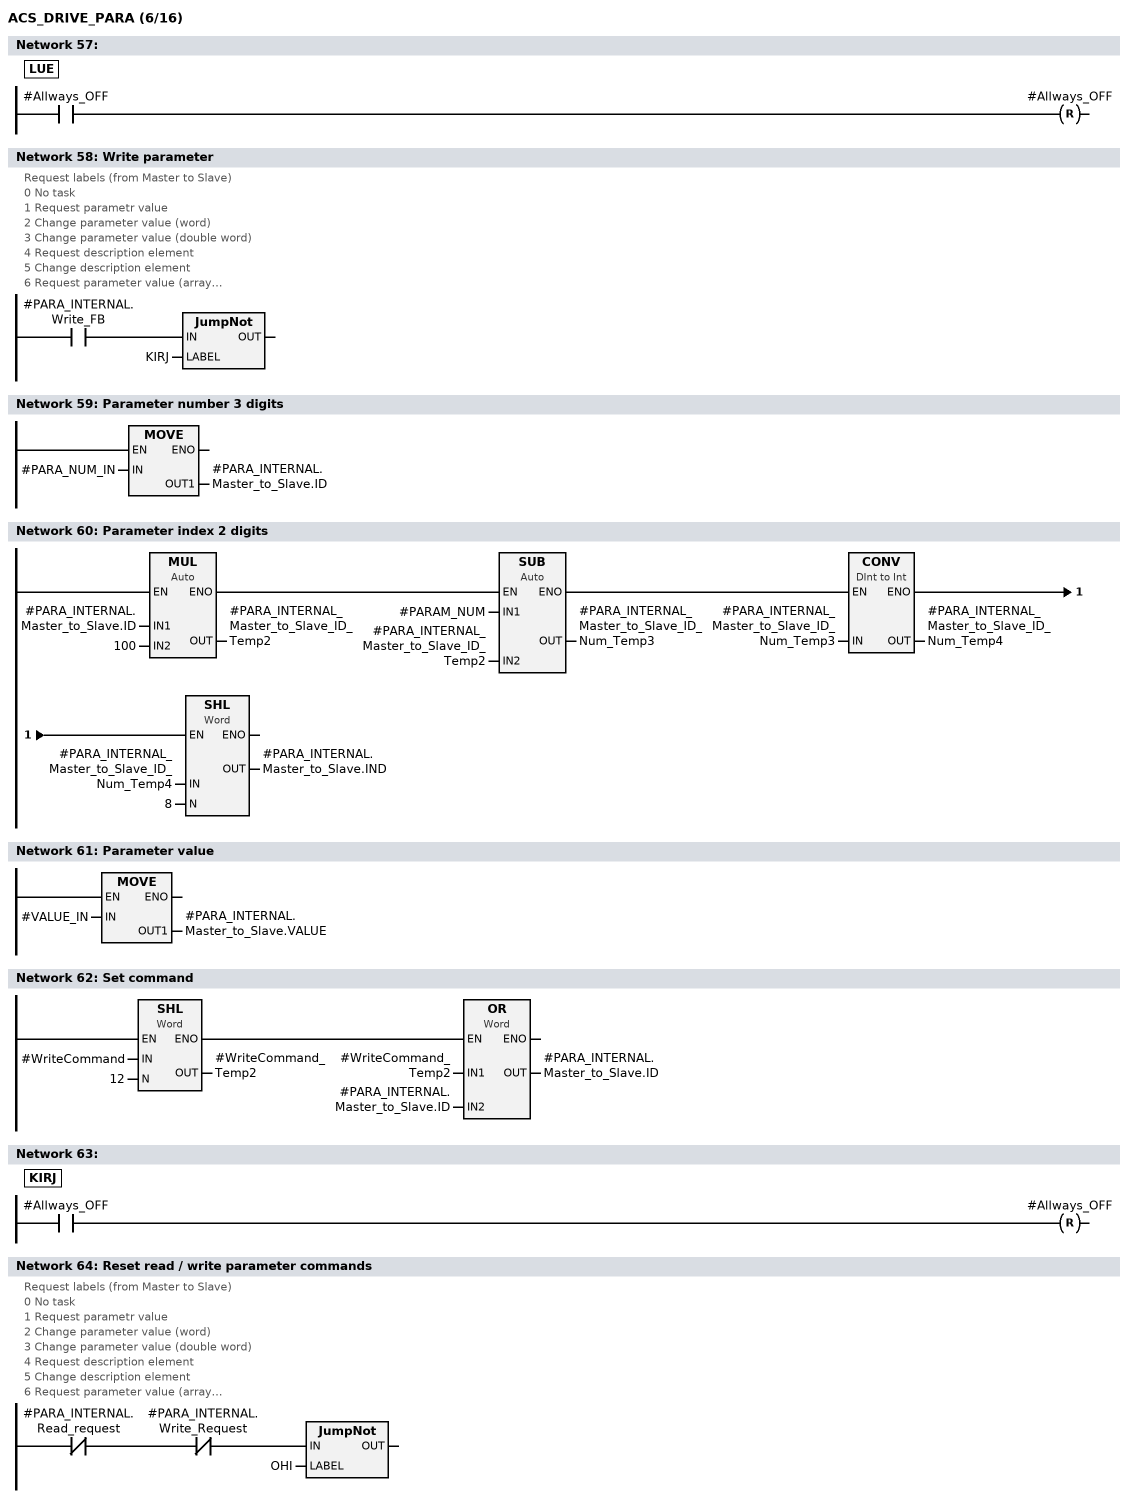
   Label( LUE )
   RUNG wire#powerrail
      Contact( #Allways_OFF )
      R_Coil( #Allways_OFF )
   END_RUNG
   // the same network as SCL:
   LUE:
   IF #Allways_OFF THEN #Allways_OFF := FALSE; END_IF;
END_REGION

REGION Network 58: Write parameter
   // Request labels (from Master to Slave)
   // 0 No task
   // 1 Request parametr value
   // 2 Change parameter value (word)
   // 3 Change parameter value (double word)
   // 4 Request description element
   // 5 Change description element
   // 6 Request parameter value (array)
   // 7 Change parameter value (array word)
   // 8 Change parameter value (array double word)
   // 9 Request number of array elements
   // 
   //  Write parameter
   // no SCL statement known for JumpNot: written as a call
   JumpNot(in := #PARA_INTERNAL.Write_FB, label := KIRJ);
END_REGION

REGION Network 59: Parameter number 3 digits
   RUNG wire#powerrail
      { S7_GenerateENO := "TRUE" } Move(in := #PARA_NUM_IN, out1 => #PARA_INTERNAL.Master_to_Slave.ID)
   END_RUNG
   // the same network as SCL:
   #PARA_INTERNAL.Master_to_Slave.ID := #PARA_NUM_IN;
END_REGION

REGION Network 60: Parameter index 2 digits
   RUNG wire#powerrail
      { S7_GenerateENO := "TRUE" } Mul(in1 := #PARA_INTERNAL.Master_to_Slave.ID, in2 := 100, out => #PARA_INTERNAL_Master_to_Slave_ID_Temp2)
      { S7_GenerateENO := "TRUE" } Sub(in1 := #PARAM_NUM, in2 := #PARA_INTERNAL_Master_to_Slave_ID_Temp2, out => #PARA_INTERNAL_Master_to_Slave_ID_Num_Temp3)
      { S7_Templates := "[SrcType := DInt, DestType := Int]"; S7_GenerateENO := "TRUE" } Convert(in := #PARA_INTERNAL_Master_to_Slave_ID_Num_Temp3, out => #PARA_INTERNAL_Master_to_Slave_ID_Num_Temp4)
      { S7_Templates := "SrcType := Word"; S7_GenerateENO := "TRUE" } Shl(in := #PARA_INTERNAL_Master_to_Slave_ID_Num_Temp4, n := 8, out => #PARA_INTERNAL.Master_to_Slave.IND)
   END_RUNG
   // the same network as SCL:
   // ENO of a box is taken as its EN; it also drops when the box reports an error
   #PARA_INTERNAL_Master_to_Slave_ID_Temp2 := #PARA_INTERNAL.Master_to_Slave.ID * 100;
   #PARA_INTERNAL_Master_to_Slave_ID_Num_Temp3 := #PARAM_NUM - #PARA_INTERNAL_Master_to_Slave_ID_Temp2;
   #PARA_INTERNAL_Master_to_Slave_ID_Num_Temp4 := DINT_TO_INT(#PARA_INTERNAL_Master_to_Slave_ID_Num_Temp3);
   #PARA_INTERNAL.Master_to_Slave.IND := SHL(IN := #PARA_INTERNAL_Master_to_Slave_ID_Num_Temp4, N := 8);
END_REGION

REGION Network 61: Parameter value
   RUNG wire#powerrail
      { S7_GenerateENO := "TRUE" } Move(in := #VALUE_IN, out1 => #PARA_INTERNAL.Master_to_Slave.VALUE)
   END_RUNG
   // the same network as SCL:
   #PARA_INTERNAL.Master_to_Slave.VALUE := #VALUE_IN;
END_REGION

REGION Network 62: Set command
   // ENO of a box is taken as its EN; it also drops when the box reports an error
   #WriteCommand_Temp2 := SHL(IN := #WriteCommand, N := 12);
   #PARA_INTERNAL.Master_to_Slave.ID := #WriteCommand_Temp2 OR #PARA_INTERNAL.Master_to_Slave.ID;
END_REGION

REGION Network 63
   Label( KIRJ )
   RUNG wire#powerrail
      Contact( #Allways_OFF )
      R_Coil( #Allways_OFF )
   END_RUNG
   // the same network as SCL:
   KIRJ:
   IF #Allways_OFF THEN #Allways_OFF := FALSE; END_IF;
END_REGION

REGION Network 64: Reset read / write parameter commands
   // Request labels (from Master to Slave)
   // 0 No task
   // 1 Request parametr value
   // 2 Change parameter value (word)
   // 3 Change parameter value (double word)
   // 4 Request description element
   // 5 Change description element
   // 6 Request parameter value (array)
   // 7 Change parameter value (array word)
   // 8 Change parameter value (array double word)
   // 9 Request number of array elements
   // 
   //  Reset parmeter commands
   // no SCL statement known for JumpNot: written as a call
   JumpNot(in := NOT #PARA_INTERNAL.Read_request AND NOT #PARA_INTERNAL.Write_Request, label := OHI);
END_REGION

REGION Network 65: Init Values
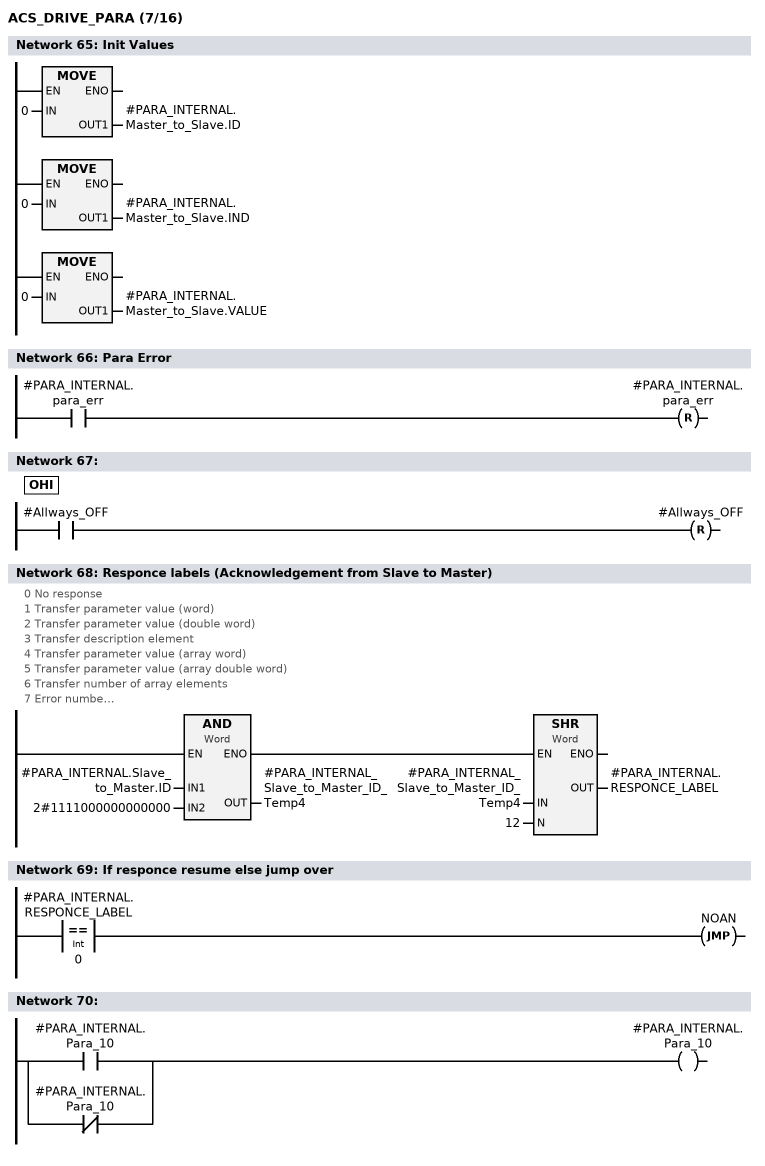
   RUNG wire#powerrail
      { S7_GenerateENO := "TRUE" } Move(in := 0, out1 => #PARA_INTERNAL.Master_to_Slave.ID)
   END_RUNG
   RUNG wire#powerrail
      { S7_GenerateENO := "TRUE" } Move(in := 0, out1 => #PARA_INTERNAL.Master_to_Slave.IND)
   END_RUNG
   RUNG wire#powerrail
      { S7_GenerateENO := "TRUE" } Move(in := 0, out1 => #PARA_INTERNAL.Master_to_Slave.VALUE)
   END_RUNG
   // the same network as SCL:
   #PARA_INTERNAL.Master_to_Slave.ID := 0;
   #PARA_INTERNAL.Master_to_Slave.IND := 0;
   #PARA_INTERNAL.Master_to_Slave.VALUE := 0;
END_REGION

REGION Network 66: Para Error
   RUNG wire#powerrail
      Contact( #PARA_INTERNAL.para_err )
      R_Coil( #PARA_INTERNAL.para_err )
   END_RUNG
   // the same network as SCL:
   IF #PARA_INTERNAL.para_err THEN #PARA_INTERNAL.para_err := FALSE; END_IF;
END_REGION

REGION Network 67
   Label( OHI )
   RUNG wire#powerrail
      Contact( #Allways_OFF )
      R_Coil( #Allways_OFF )
   END_RUNG
   // the same network as SCL:
   OHI:
   IF #Allways_OFF THEN #Allways_OFF := FALSE; END_IF;
END_REGION

REGION Network 68: Responce labels (Acknowledgement from Slave to Master)
   // 0 No response
   // 1 Transfer parameter value (word)
   // 2 Transfer parameter value (double word)
   // 3 Transfer description element
   // 4 Transfer parameter value (array word)
   // 5 Transfer parameter value (array double word)
   // 6 Transfer number of array elements
   // 7 Error number
   // - 0 Illegal parameter number
   // - 1 Parameter value cannot be changed
   // - 2 Lower or upper limit violated
   // - 3 Error subindex
   // - 4 No array
   // - 5 Incorrect data type
   // - 6 Setting not allowed (can only be reset)
   // - 7 Descriptive element cannot be changed
   // - 9 Descriptive data not available
   // - 11 No parameter change rights
   // - 15 Text array not available
   // - 17 Task cannot be executed due to operating status
   // - 18 Other error
   // - 101 Vendor specific
   // - 102 Request not supported
   // - 103 Request cannot be compeleted due to communication error
   // - 110 Failure during write to non-volatile memory
   // - 111 Request aborted due to time-out
   // - 120 Parameter cannot be mapped to PZD
   // - 121 Parameter cannot be mapped to PZD (end of memory)
   // - 122 Parameter cannot be mapped to PZD (multiple PZD write)
   // - 130 Cannot map Control Word bit (parameter 933-937)
   // - 140 Cannot change mode to TORGUE
   // - 150 Internal buffer overflow
   // - 160 Internal communication error
   // 8 No parameter change rights for PKW interface
   // 9 Parameter data signal (word)
   // 10 Parameter data signal (double word)
   //  Mask responce labels
   RUNG wire#powerrail
      { S7_Templates := "SrcType := Word"; S7_GenerateENO := "TRUE" } And(in1 := #PARA_INTERNAL.Slave_to_Master.ID, in2 := 2#1111000000000000, out => #PARA_INTERNAL_Slave_to_Master_ID_Temp4)
      { S7_Templates := "SrcType := Word"; S7_GenerateENO := "TRUE" } Shr(in := #PARA_INTERNAL_Slave_to_Master_ID_Temp4, n := 12, out => #PARA_INTERNAL.RESPONCE_LABEL)
   END_RUNG
   // the same network as SCL:
   #PARA_INTERNAL_Slave_to_Master_ID_Temp4 := #PARA_INTERNAL.Slave_to_Master.ID AND 2#1111000000000000;
   #PARA_INTERNAL.RESPONCE_LABEL := SHR(IN := #PARA_INTERNAL_Slave_to_Master_ID_Temp4, N := 12);
END_REGION

REGION Network 69: If responce resume else jump over
   RUNG wire#powerrail
      { S7_Templates := "SrcType := Int" } EQ_Contact(in1 := #PARA_INTERNAL.RESPONCE_LABEL, in2 := 0)
      JumpCoil( NOAN )
   END_RUNG
   // the same network as SCL:
   IF #PARA_INTERNAL.RESPONCE_LABEL = 0 THEN GOTO NOAN; END_IF;
END_REGION

REGION Network 70
   RUNG wire#powerrail
      Contact( #PARA_INTERNAL.Para_10 )
      wire#w1
      Coil( #PARA_INTERNAL.Para_10 )
   END_RUNG
   RUNG wire#powerrail
      I_Contact( #PARA_INTERNAL.Para_10 )
   END_RUNG wire#w1
   // the same network as SCL:
   #PARA_INTERNAL.Para_10 := #PARA_INTERNAL.Para_10 OR NOT #PARA_INTERNAL.Para_10;
END_REGION

REGION Network 71: Update responce parameter and index to output
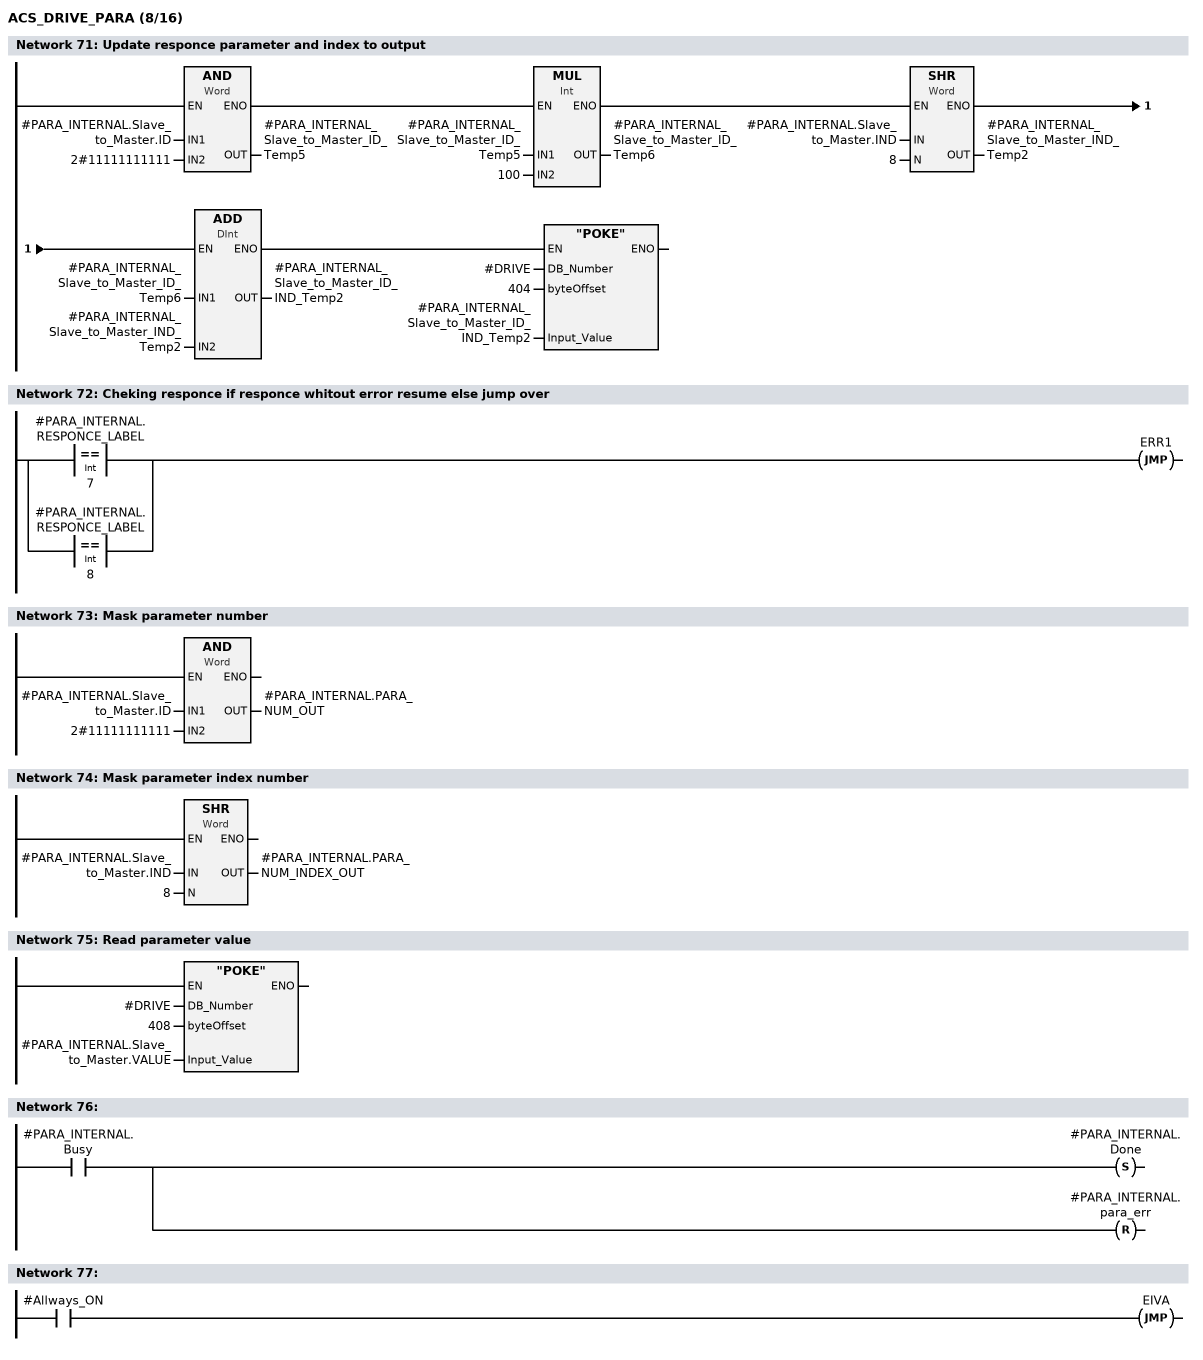
   RUNG wire#powerrail
      { S7_Templates := "SrcType := Word"; S7_GenerateENO := "TRUE" } And(in1 := #PARA_INTERNAL.Slave_to_Master.ID, in2 := 2#11111111111, out => #PARA_INTERNAL_Slave_to_Master_ID_Temp5)
      { S7_Templates := "SrcType := Int"; S7_GenerateENO := "TRUE" } Mul(in1 := #PARA_INTERNAL_Slave_to_Master_ID_Temp5, in2 := 100, out => #PARA_INTERNAL_Slave_to_Master_ID_Temp6)
      { S7_Templates := "SrcType := Word"; S7_GenerateENO := "TRUE" } Shr(in := #PARA_INTERNAL.Slave_to_Master.IND, n := 8, out => #PARA_INTERNAL_Slave_to_Master_IND_Temp2)
      { S7_Templates := "SrcType := DInt"; S7_GenerateENO := "TRUE" } Add(in1 := #PARA_INTERNAL_Slave_to_Master_ID_Temp6, in2 := #PARA_INTERNAL_Slave_to_Master_IND_Temp2, out => #PARA_INTERNAL_Slave_to_Master_ID_IND_Temp2)
      "POKE"(DB_Number := #DRIVE, byteOffset := 404, Input_Value := #PARA_INTERNAL_Slave_to_Master_ID_IND_Temp2)
   END_RUNG
   // the same network as SCL:
   // ENO of a box is taken as its EN; it also drops when the box reports an error
   #PARA_INTERNAL_Slave_to_Master_ID_Temp5 := #PARA_INTERNAL.Slave_to_Master.ID AND 2#11111111111;
   #PARA_INTERNAL_Slave_to_Master_ID_Temp6 := #PARA_INTERNAL_Slave_to_Master_ID_Temp5 * 100;
   #PARA_INTERNAL_Slave_to_Master_IND_Temp2 := SHR(IN := #PARA_INTERNAL.Slave_to_Master.IND, N := 8);
   #PARA_INTERNAL_Slave_to_Master_ID_IND_Temp2 := #PARA_INTERNAL_Slave_to_Master_ID_Temp6 + #PARA_INTERNAL_Slave_to_Master_IND_Temp2;
   "POKE"(DB_Number := #DRIVE, byteOffset := 404, Input_Value := #PARA_INTERNAL_Slave_to_Master_ID_IND_Temp2);
END_REGION

REGION Network 72: Cheking responce if responce whitout error resume else jump over
   RUNG wire#powerrail
      { S7_Templates := "SrcType := Int" } EQ_Contact(in1 := #PARA_INTERNAL.RESPONCE_LABEL, in2 := 7)
      wire#w1
      JumpCoil( ERR1 )
   END_RUNG
   RUNG wire#powerrail
      { S7_Templates := "SrcType := Int" } EQ_Contact(in1 := #PARA_INTERNAL.RESPONCE_LABEL, in2 := 8)
   END_RUNG wire#w1
   // the same network as SCL:
   IF (#PARA_INTERNAL.RESPONCE_LABEL = 7) OR (#PARA_INTERNAL.RESPONCE_LABEL = 8) THEN GOTO ERR1; END_IF;
END_REGION

REGION Network 73: Mask parameter number
   RUNG wire#powerrail
      { S7_Templates := "SrcType := Word"; S7_GenerateENO := "TRUE" } And(in1 := #PARA_INTERNAL.Slave_to_Master.ID, in2 := 2#11111111111, out => #PARA_INTERNAL.PARA_NUM_OUT)
   END_RUNG
   // the same network as SCL:
   #PARA_INTERNAL.PARA_NUM_OUT := #PARA_INTERNAL.Slave_to_Master.ID AND 2#11111111111;
END_REGION

REGION Network 74: Mask parameter index number
   RUNG wire#powerrail
      { S7_Templates := "SrcType := Word"; S7_GenerateENO := "TRUE" } Shr(in := #PARA_INTERNAL.Slave_to_Master.IND, n := 8, out => #PARA_INTERNAL.PARA_NUM_INDEX_OUT)
   END_RUNG
   // the same network as SCL:
   #PARA_INTERNAL.PARA_NUM_INDEX_OUT := SHR(IN := #PARA_INTERNAL.Slave_to_Master.IND, N := 8);
END_REGION

REGION Network 75: Read parameter value
   RUNG wire#powerrail
      "POKE"(DB_Number := #DRIVE, byteOffset := 408, Input_Value := #PARA_INTERNAL.Slave_to_Master.VALUE)
   END_RUNG
   // the same network as SCL:
   "POKE"(DB_Number := #DRIVE, byteOffset := 408, Input_Value := #PARA_INTERNAL.Slave_to_Master.VALUE);
END_REGION

REGION Network 76
   RUNG wire#powerrail
      Contact( #PARA_INTERNAL.Busy )
      wire#w1
      S_Coil( #PARA_INTERNAL.Done )
   END_RUNG
   RUNG wire#w1
      R_Coil( #PARA_INTERNAL.para_err )
   END_RUNG
   // the same network as SCL:
   IF #PARA_INTERNAL.Busy THEN
       #PARA_INTERNAL.Done := TRUE;
       #PARA_INTERNAL.para_err := FALSE;
   END_IF;
END_REGION

REGION Network 77
   RUNG wire#powerrail
      Contact( #Allways_ON )
      JumpCoil( EIVA )
   END_RUNG
   // the same network as SCL:
   IF #Allways_ON THEN GOTO EIVA; END_IF;
END_REGION

REGION Network 78: Error handlin in responce code
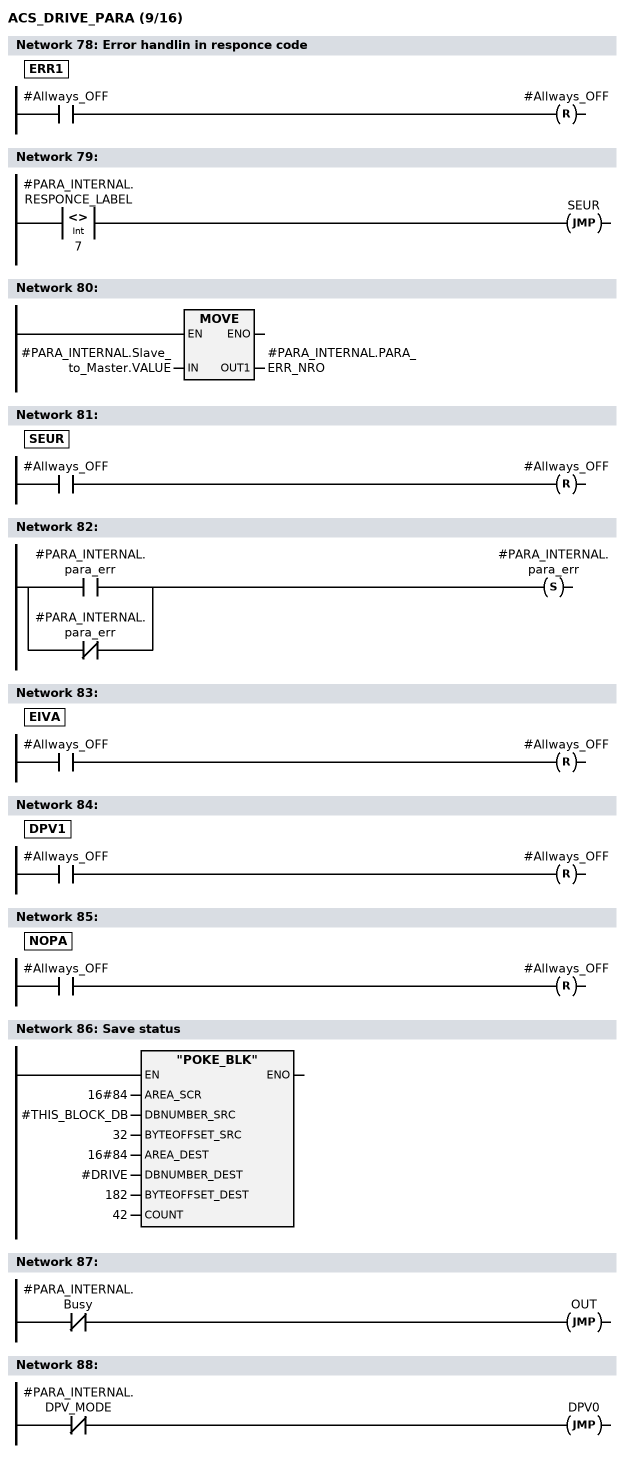
   Label( ERR1 )
   RUNG wire#powerrail
      Contact( #Allways_OFF )
      R_Coil( #Allways_OFF )
   END_RUNG
   // the same network as SCL:
   ERR1:
   IF #Allways_OFF THEN #Allways_OFF := FALSE; END_IF;
END_REGION

REGION Network 79
   RUNG wire#powerrail
      { S7_Templates := "SrcType := Int" } NE_Contact(in1 := #PARA_INTERNAL.RESPONCE_LABEL, in2 := 7)
      JumpCoil( SEUR )
   END_RUNG
   // the same network as SCL:
   IF #PARA_INTERNAL.RESPONCE_LABEL <> 7 THEN GOTO SEUR; END_IF;
END_REGION

REGION Network 80
   RUNG wire#powerrail
      { S7_GenerateENO := "TRUE" } Move(in := #PARA_INTERNAL.Slave_to_Master.VALUE, out1 => #PARA_INTERNAL.PARA_ERR_NRO)
   END_RUNG
   // the same network as SCL:
   #PARA_INTERNAL.PARA_ERR_NRO := #PARA_INTERNAL.Slave_to_Master.VALUE;
END_REGION

REGION Network 81
   Label( SEUR )
   RUNG wire#powerrail
      Contact( #Allways_OFF )
      R_Coil( #Allways_OFF )
   END_RUNG
   // the same network as SCL:
   SEUR:
   IF #Allways_OFF THEN #Allways_OFF := FALSE; END_IF;
END_REGION

REGION Network 82
   RUNG wire#powerrail
      Contact( #PARA_INTERNAL.para_err )
      wire#w1
      S_Coil( #PARA_INTERNAL.para_err )
   END_RUNG
   RUNG wire#powerrail
      I_Contact( #PARA_INTERNAL.para_err )
   END_RUNG wire#w1
   // the same network as SCL:
   IF #PARA_INTERNAL.para_err OR NOT #PARA_INTERNAL.para_err THEN #PARA_INTERNAL.para_err := TRUE; END_IF;
END_REGION

REGION Network 83
   Label( EIVA )
   RUNG wire#powerrail
      Contact( #Allways_OFF )
      R_Coil( #Allways_OFF )
   END_RUNG
   // the same network as SCL:
   EIVA:
   IF #Allways_OFF THEN #Allways_OFF := FALSE; END_IF;
END_REGION

REGION Network 84
   Label( DPV1 )
   RUNG wire#powerrail
      Contact( #Allways_OFF )
      R_Coil( #Allways_OFF )
   END_RUNG
   // the same network as SCL:
   DPV1:
   IF #Allways_OFF THEN #Allways_OFF := FALSE; END_IF;
END_REGION

REGION Network 85
   Label( NOPA )
   RUNG wire#powerrail
      Contact( #Allways_OFF )
      R_Coil( #Allways_OFF )
   END_RUNG
   // the same network as SCL:
   NOPA:
   IF #Allways_OFF THEN #Allways_OFF := FALSE; END_IF;
END_REGION

REGION Network 86: Save status
   RUNG wire#powerrail
      "POKE_BLK"(AREA_SCR := 16#84, DBNUMBER_SRC := #THIS_BLOCK_DB, BYTEOFFSET_SRC := 32, AREA_DEST := 16#84, DBNUMBER_DEST := #DRIVE, BYTEOFFSET_DEST := 182, COUNT := 42)
   END_RUNG
   // the same network as SCL:
   "POKE_BLK"(AREA_SCR := 16#84,
              DBNUMBER_SRC := #THIS_BLOCK_DB,
              BYTEOFFSET_SRC := 32,
              AREA_DEST := 16#84,
              DBNUMBER_DEST := #DRIVE,
              BYTEOFFSET_DEST := 182,
              COUNT := 42);
END_REGION

REGION Network 87
   RUNG wire#powerrail
      I_Contact( #PARA_INTERNAL.Busy )
      JumpCoil( OUT )
   END_RUNG
   // the same network as SCL:
   IF NOT #PARA_INTERNAL.Busy THEN GOTO OUT; END_IF;
END_REGION

REGION Network 88
   RUNG wire#powerrail
      I_Contact( #PARA_INTERNAL.DPV_MODE )
      JumpCoil( DPV0 )
   END_RUNG
   // the same network as SCL:
   IF NOT #PARA_INTERNAL.DPV_MODE THEN GOTO DPV0; END_IF;
END_REGION

REGION Network 89
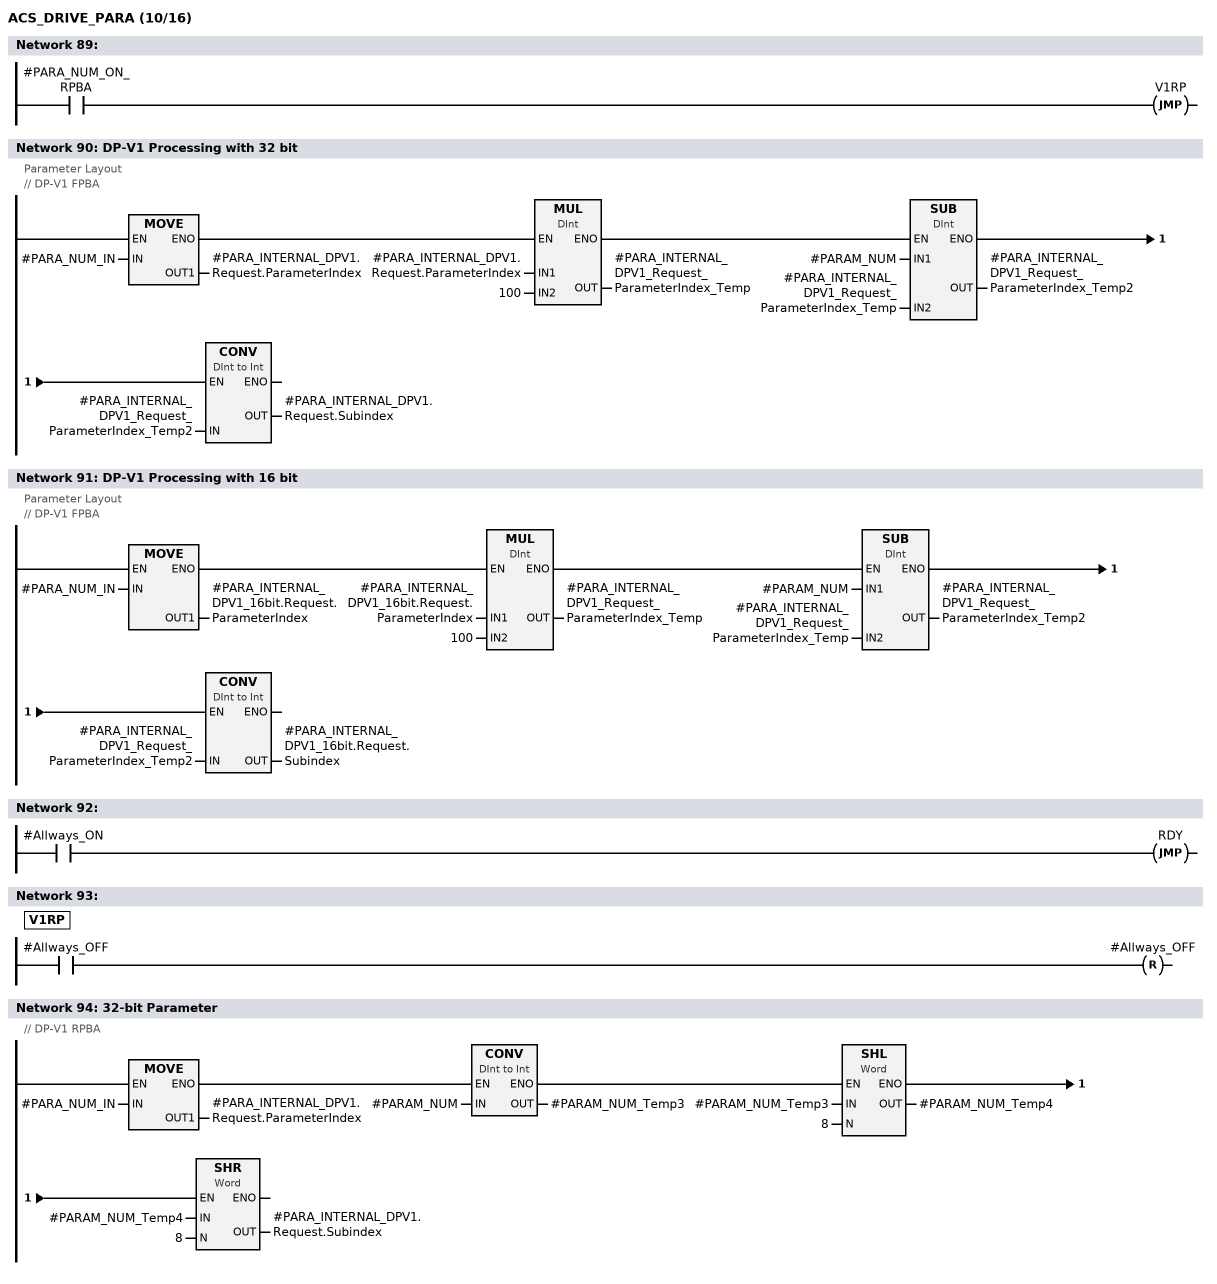
   RUNG wire#powerrail
      Contact( #PARA_NUM_ON_RPBA )
      JumpCoil( V1RP )
   END_RUNG
   // the same network as SCL:
   IF #PARA_NUM_ON_RPBA THEN GOTO V1RP; END_IF;
END_REGION

REGION Network 90: DP-V1 Processing with 32 bit
   // Parameter Layout
   //  // DP-V1 FPBA
   RUNG wire#powerrail
      { S7_GenerateENO := "TRUE" } Move(in := #PARA_NUM_IN, out1 => #PARA_INTERNAL_DPV1.Request.ParameterIndex)
      { S7_Templates := "SrcType := DInt"; S7_GenerateENO := "TRUE" } Mul(in1 := #PARA_INTERNAL_DPV1.Request.ParameterIndex, in2 := 100, out => #PARA_INTERNAL_DPV1_Request_ParameterIndex_Temp)
      { S7_Templates := "SrcType := DInt"; S7_GenerateENO := "TRUE" } Sub(in1 := #PARAM_NUM, in2 := #PARA_INTERNAL_DPV1_Request_ParameterIndex_Temp, out => #PARA_INTERNAL_DPV1_Request_ParameterIndex_Temp2)
      { S7_Templates := "[SrcType := DInt, DestType := Int]"; S7_GenerateENO := "TRUE" } Convert(in := #PARA_INTERNAL_DPV1_Request_ParameterIndex_Temp2, out => #PARA_INTERNAL_DPV1.Request.Subindex)
   END_RUNG
   // the same network as SCL:
   // ENO of a box is taken as its EN; it also drops when the box reports an error
   #PARA_INTERNAL_DPV1.Request.ParameterIndex := #PARA_NUM_IN;
   #PARA_INTERNAL_DPV1_Request_ParameterIndex_Temp := #PARA_INTERNAL_DPV1.Request.ParameterIndex * 100;
   #PARA_INTERNAL_DPV1_Request_ParameterIndex_Temp2 := #PARAM_NUM - #PARA_INTERNAL_DPV1_Request_ParameterIndex_Temp;
   #PARA_INTERNAL_DPV1.Request.Subindex := DINT_TO_INT(#PARA_INTERNAL_DPV1_Request_ParameterIndex_Temp2);
END_REGION

REGION Network 91: DP-V1 Processing with 16 bit
   // Parameter Layout
   //  // DP-V1 FPBA
   RUNG wire#powerrail
      { S7_GenerateENO := "TRUE" } Move(in := #PARA_NUM_IN, out1 => #PARA_INTERNAL_DPV1_16bit.Request.ParameterIndex)
      { S7_Templates := "SrcType := DInt"; S7_GenerateENO := "TRUE" } Mul(in1 := #PARA_INTERNAL_DPV1_16bit.Request.ParameterIndex, in2 := 100, out => #PARA_INTERNAL_DPV1_Request_ParameterIndex_Temp)
      { S7_Templates := "SrcType := DInt"; S7_GenerateENO := "TRUE" } Sub(in1 := #PARAM_NUM, in2 := #PARA_INTERNAL_DPV1_Request_ParameterIndex_Temp, out => #PARA_INTERNAL_DPV1_Request_ParameterIndex_Temp2)
      { S7_Templates := "[SrcType := DInt, DestType := Int]"; S7_GenerateENO := "TRUE" } Convert(in := #PARA_INTERNAL_DPV1_Request_ParameterIndex_Temp2, out => #PARA_INTERNAL_DPV1_16bit.Request.Subindex)
   END_RUNG
   // the same network as SCL:
   // ENO of a box is taken as its EN; it also drops when the box reports an error
   #PARA_INTERNAL_DPV1_16bit.Request.ParameterIndex := #PARA_NUM_IN;
   #PARA_INTERNAL_DPV1_Request_ParameterIndex_Temp := #PARA_INTERNAL_DPV1_16bit.Request.ParameterIndex * 100;
   #PARA_INTERNAL_DPV1_Request_ParameterIndex_Temp2 := #PARAM_NUM - #PARA_INTERNAL_DPV1_Request_ParameterIndex_Temp;
   #PARA_INTERNAL_DPV1_16bit.Request.Subindex := DINT_TO_INT(#PARA_INTERNAL_DPV1_Request_ParameterIndex_Temp2);
END_REGION

REGION Network 92
   RUNG wire#powerrail
      Contact( #Allways_ON )
      JumpCoil( RDY )
   END_RUNG
   // the same network as SCL:
   IF #Allways_ON THEN GOTO RDY; END_IF;
END_REGION

REGION Network 93
   Label( V1RP )
   RUNG wire#powerrail
      Contact( #Allways_OFF )
      R_Coil( #Allways_OFF )
   END_RUNG
   // the same network as SCL:
   V1RP:
   IF #Allways_OFF THEN #Allways_OFF := FALSE; END_IF;
END_REGION

REGION Network 94: 32-bit Parameter
   // // DP-V1 RPBA
   RUNG wire#powerrail
      { S7_GenerateENO := "TRUE" } Move(in := #PARA_NUM_IN, out1 => #PARA_INTERNAL_DPV1.Request.ParameterIndex)
      { S7_Templates := "[SrcType := DInt, DestType := Int]"; S7_GenerateENO := "TRUE" } Convert(in := #PARAM_NUM, out => #PARAM_NUM_Temp3)
      { S7_Templates := "SrcType := Word"; S7_GenerateENO := "TRUE" } Shl(in := #PARAM_NUM_Temp3, n := 8, out => #PARAM_NUM_Temp4)
      { S7_Templates := "SrcType := Word"; S7_GenerateENO := "TRUE" } Shr(in := #PARAM_NUM_Temp4, n := 8, out => #PARA_INTERNAL_DPV1.Request.Subindex)
   END_RUNG
   // the same network as SCL:
   // ENO of a box is taken as its EN; it also drops when the box reports an error
   #PARA_INTERNAL_DPV1.Request.ParameterIndex := #PARA_NUM_IN;
   #PARAM_NUM_Temp3 := DINT_TO_INT(#PARAM_NUM);
   #PARAM_NUM_Temp4 := SHL(IN := #PARAM_NUM_Temp3, N := 8);
   #PARA_INTERNAL_DPV1.Request.Subindex := SHR(IN := #PARAM_NUM_Temp4, N := 8);
END_REGION

REGION Network 95: 16-bit Parameter
   // // DP-V1 RPBA
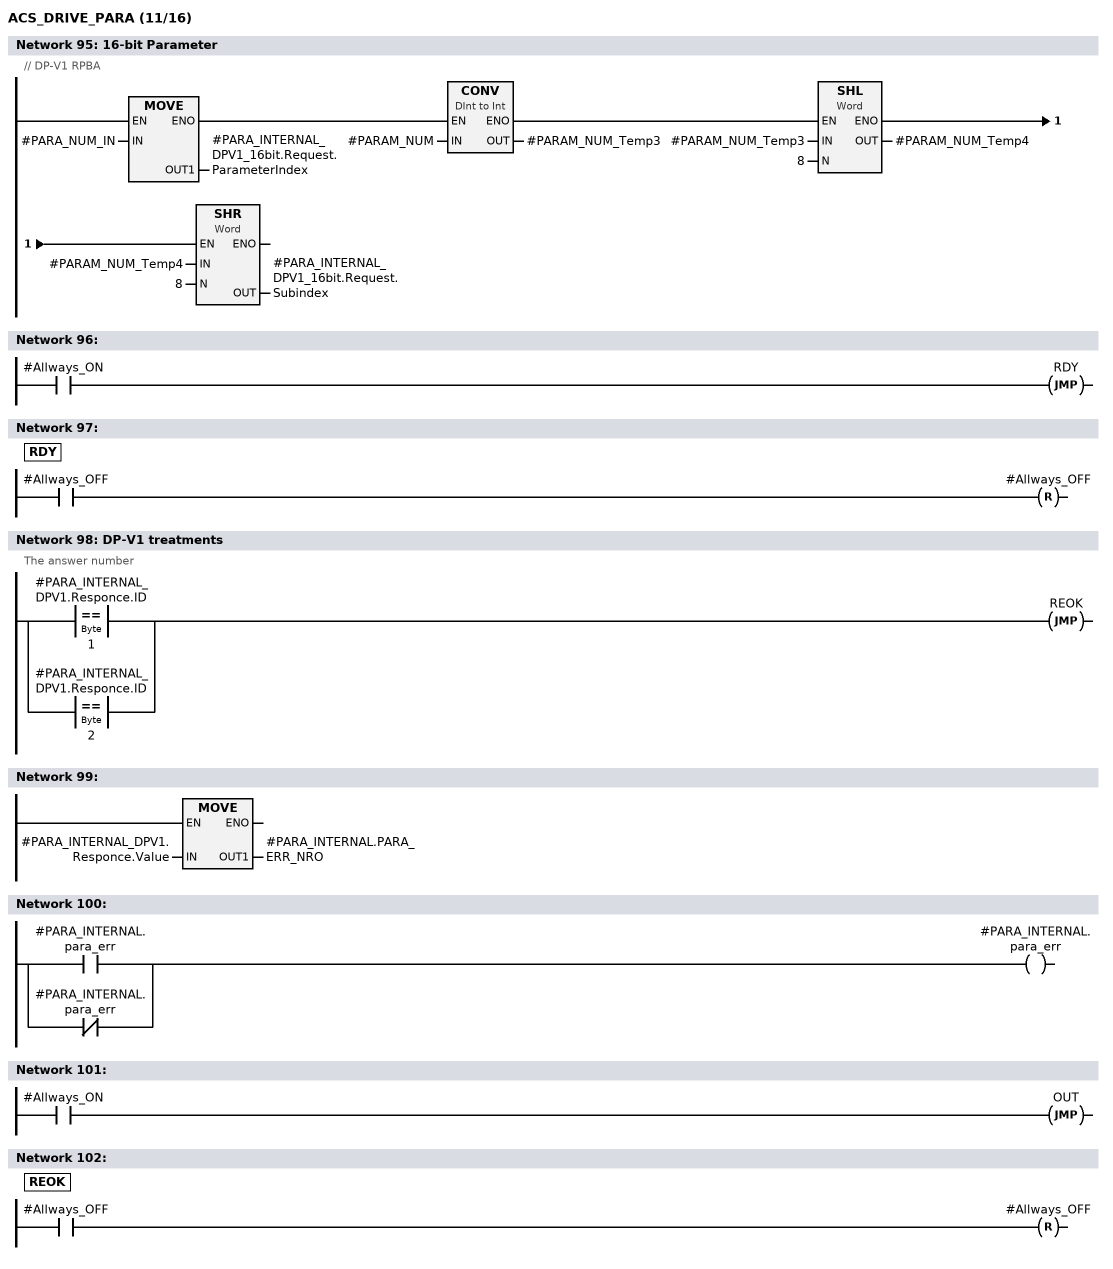
   RUNG wire#powerrail
      { S7_GenerateENO := "TRUE" } Move(in := #PARA_NUM_IN, out1 => #PARA_INTERNAL_DPV1_16bit.Request.ParameterIndex)
      { S7_Templates := "[SrcType := DInt, DestType := Int]"; S7_GenerateENO := "TRUE" } Convert(in := #PARAM_NUM, out => #PARAM_NUM_Temp3)
      { S7_Templates := "SrcType := Word"; S7_GenerateENO := "TRUE" } Shl(in := #PARAM_NUM_Temp3, n := 8, out => #PARAM_NUM_Temp4)
      { S7_Templates := "SrcType := Word"; S7_GenerateENO := "TRUE" } Shr(in := #PARAM_NUM_Temp4, n := 8, out => #PARA_INTERNAL_DPV1_16bit.Request.Subindex)
   END_RUNG
   // the same network as SCL:
   // ENO of a box is taken as its EN; it also drops when the box reports an error
   #PARA_INTERNAL_DPV1_16bit.Request.ParameterIndex := #PARA_NUM_IN;
   #PARAM_NUM_Temp3 := DINT_TO_INT(#PARAM_NUM);
   #PARAM_NUM_Temp4 := SHL(IN := #PARAM_NUM_Temp3, N := 8);
   #PARA_INTERNAL_DPV1_16bit.Request.Subindex := SHR(IN := #PARAM_NUM_Temp4, N := 8);
END_REGION

REGION Network 96
   RUNG wire#powerrail
      Contact( #Allways_ON )
      JumpCoil( RDY )
   END_RUNG
   // the same network as SCL:
   IF #Allways_ON THEN GOTO RDY; END_IF;
END_REGION

REGION Network 97
   Label( RDY )
   RUNG wire#powerrail
      Contact( #Allways_OFF )
      R_Coil( #Allways_OFF )
   END_RUNG
   // the same network as SCL:
   RDY:
   IF #Allways_OFF THEN #Allways_OFF := FALSE; END_IF;
END_REGION

REGION Network 98: DP-V1 treatments
   // The answer number
   RUNG wire#powerrail
      { S7_Templates := "SrcType := Byte" } EQ_Contact(in1 := #PARA_INTERNAL_DPV1.Responce.ID, in2 := 1)
      wire#w1
      JumpCoil( REOK )
   END_RUNG
   RUNG wire#powerrail
      { S7_Templates := "SrcType := Byte" } EQ_Contact(in1 := #PARA_INTERNAL_DPV1.Responce.ID, in2 := 2)
   END_RUNG wire#w1
   // the same network as SCL:
   IF (#PARA_INTERNAL_DPV1.Responce.ID = 1) OR (#PARA_INTERNAL_DPV1.Responce.ID = 2) THEN GOTO REOK; END_IF;
END_REGION

REGION Network 99
   RUNG wire#powerrail
      { S7_GenerateENO := "TRUE" } Move(in := #PARA_INTERNAL_DPV1.Responce.Value, out1 => #PARA_INTERNAL.PARA_ERR_NRO)
   END_RUNG
   // the same network as SCL:
   #PARA_INTERNAL.PARA_ERR_NRO := #PARA_INTERNAL_DPV1.Responce.Value;
END_REGION

REGION Network 100
   RUNG wire#powerrail
      Contact( #PARA_INTERNAL.para_err )
      wire#w1
      Coil( #PARA_INTERNAL.para_err )
   END_RUNG
   RUNG wire#powerrail
      I_Contact( #PARA_INTERNAL.para_err )
   END_RUNG wire#w1
   // the same network as SCL:
   #PARA_INTERNAL.para_err := #PARA_INTERNAL.para_err OR NOT #PARA_INTERNAL.para_err;
END_REGION

REGION Network 101
   RUNG wire#powerrail
      Contact( #Allways_ON )
      JumpCoil( OUT )
   END_RUNG
   // the same network as SCL:
   IF #Allways_ON THEN GOTO OUT; END_IF;
END_REGION

REGION Network 102
   Label( REOK )
   RUNG wire#powerrail
      Contact( #Allways_OFF )
      R_Coil( #Allways_OFF )
   END_RUNG
   // the same network as SCL:
   REOK:
   IF #Allways_OFF THEN #Allways_OFF := FALSE; END_IF;
END_REGION

REGION Network 103
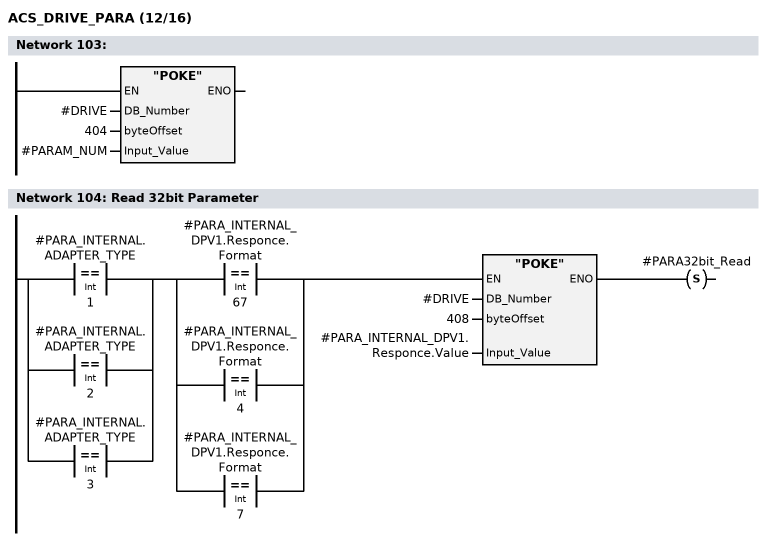
   RUNG wire#powerrail
      "POKE"(DB_Number := #DRIVE, byteOffset := 404, Input_Value := #PARAM_NUM)
   END_RUNG
   // the same network as SCL:
   "POKE"(DB_Number := #DRIVE, byteOffset := 404, Input_Value := #PARAM_NUM);
END_REGION

REGION Network 104: Read 32bit Parameter
   RUNG wire#powerrail
      { S7_Templates := "SrcType := Int" } EQ_Contact(in1 := #PARA_INTERNAL.ADAPTER_TYPE, in2 := 1)
      wire#w1
      { S7_Templates := "SrcType := Int" } EQ_Contact(in1 := #PARA_INTERNAL_DPV1.Responce.Format, in2 := 67)
      wire#w2
      "POKE"(DB_Number := #DRIVE, byteOffset := 408, Input_Value := #PARA_INTERNAL_DPV1.Responce.Value)
      S_Coil( #PARA32bit_Read )
   END_RUNG
   RUNG wire#powerrail
      { S7_Templates := "SrcType := Int" } EQ_Contact(in1 := #PARA_INTERNAL.ADAPTER_TYPE, in2 := 2)
   END_RUNG wire#w1
   RUNG wire#powerrail
      { S7_Templates := "SrcType := Int" } EQ_Contact(in1 := #PARA_INTERNAL.ADAPTER_TYPE, in2 := 3)
   END_RUNG wire#w1
   RUNG wire#w1
      { S7_Templates := "SrcType := Int" } EQ_Contact(in1 := #PARA_INTERNAL_DPV1.Responce.Format, in2 := 4)
   END_RUNG wire#w2
   RUNG wire#w1
      { S7_Templates := "SrcType := Int" } EQ_Contact(in1 := #PARA_INTERNAL_DPV1.Responce.Format, in2 := 7)
   END_RUNG wire#w2
   // the same network as SCL:
   "POKE"(EN := ((#PARA_INTERNAL.ADAPTER_TYPE = 1) OR (#PARA_INTERNAL.ADAPTER_TYPE = 2) OR (#PARA_INTERNAL.ADAPTER_TYPE = 3)) AND ((#PARA_INTERNAL_DPV1.Responce.Format = 67) OR (#PARA_INTERNAL_DPV1.Responce.Format = 4) OR (#PARA_INTERNAL_DPV1.Responce.Format = 7)),
          DB_Number := #DRIVE,
          byteOffset := 408,
          Input_Value := #PARA_INTERNAL_DPV1.Responce.Value,
          ENO => #_w1);
   IF #_w1 THEN #PARA32bit_Read := TRUE; END_IF;
END_REGION

REGION Network 105: Read 16bit Parameter: Swap Responce Value from DWord to Word
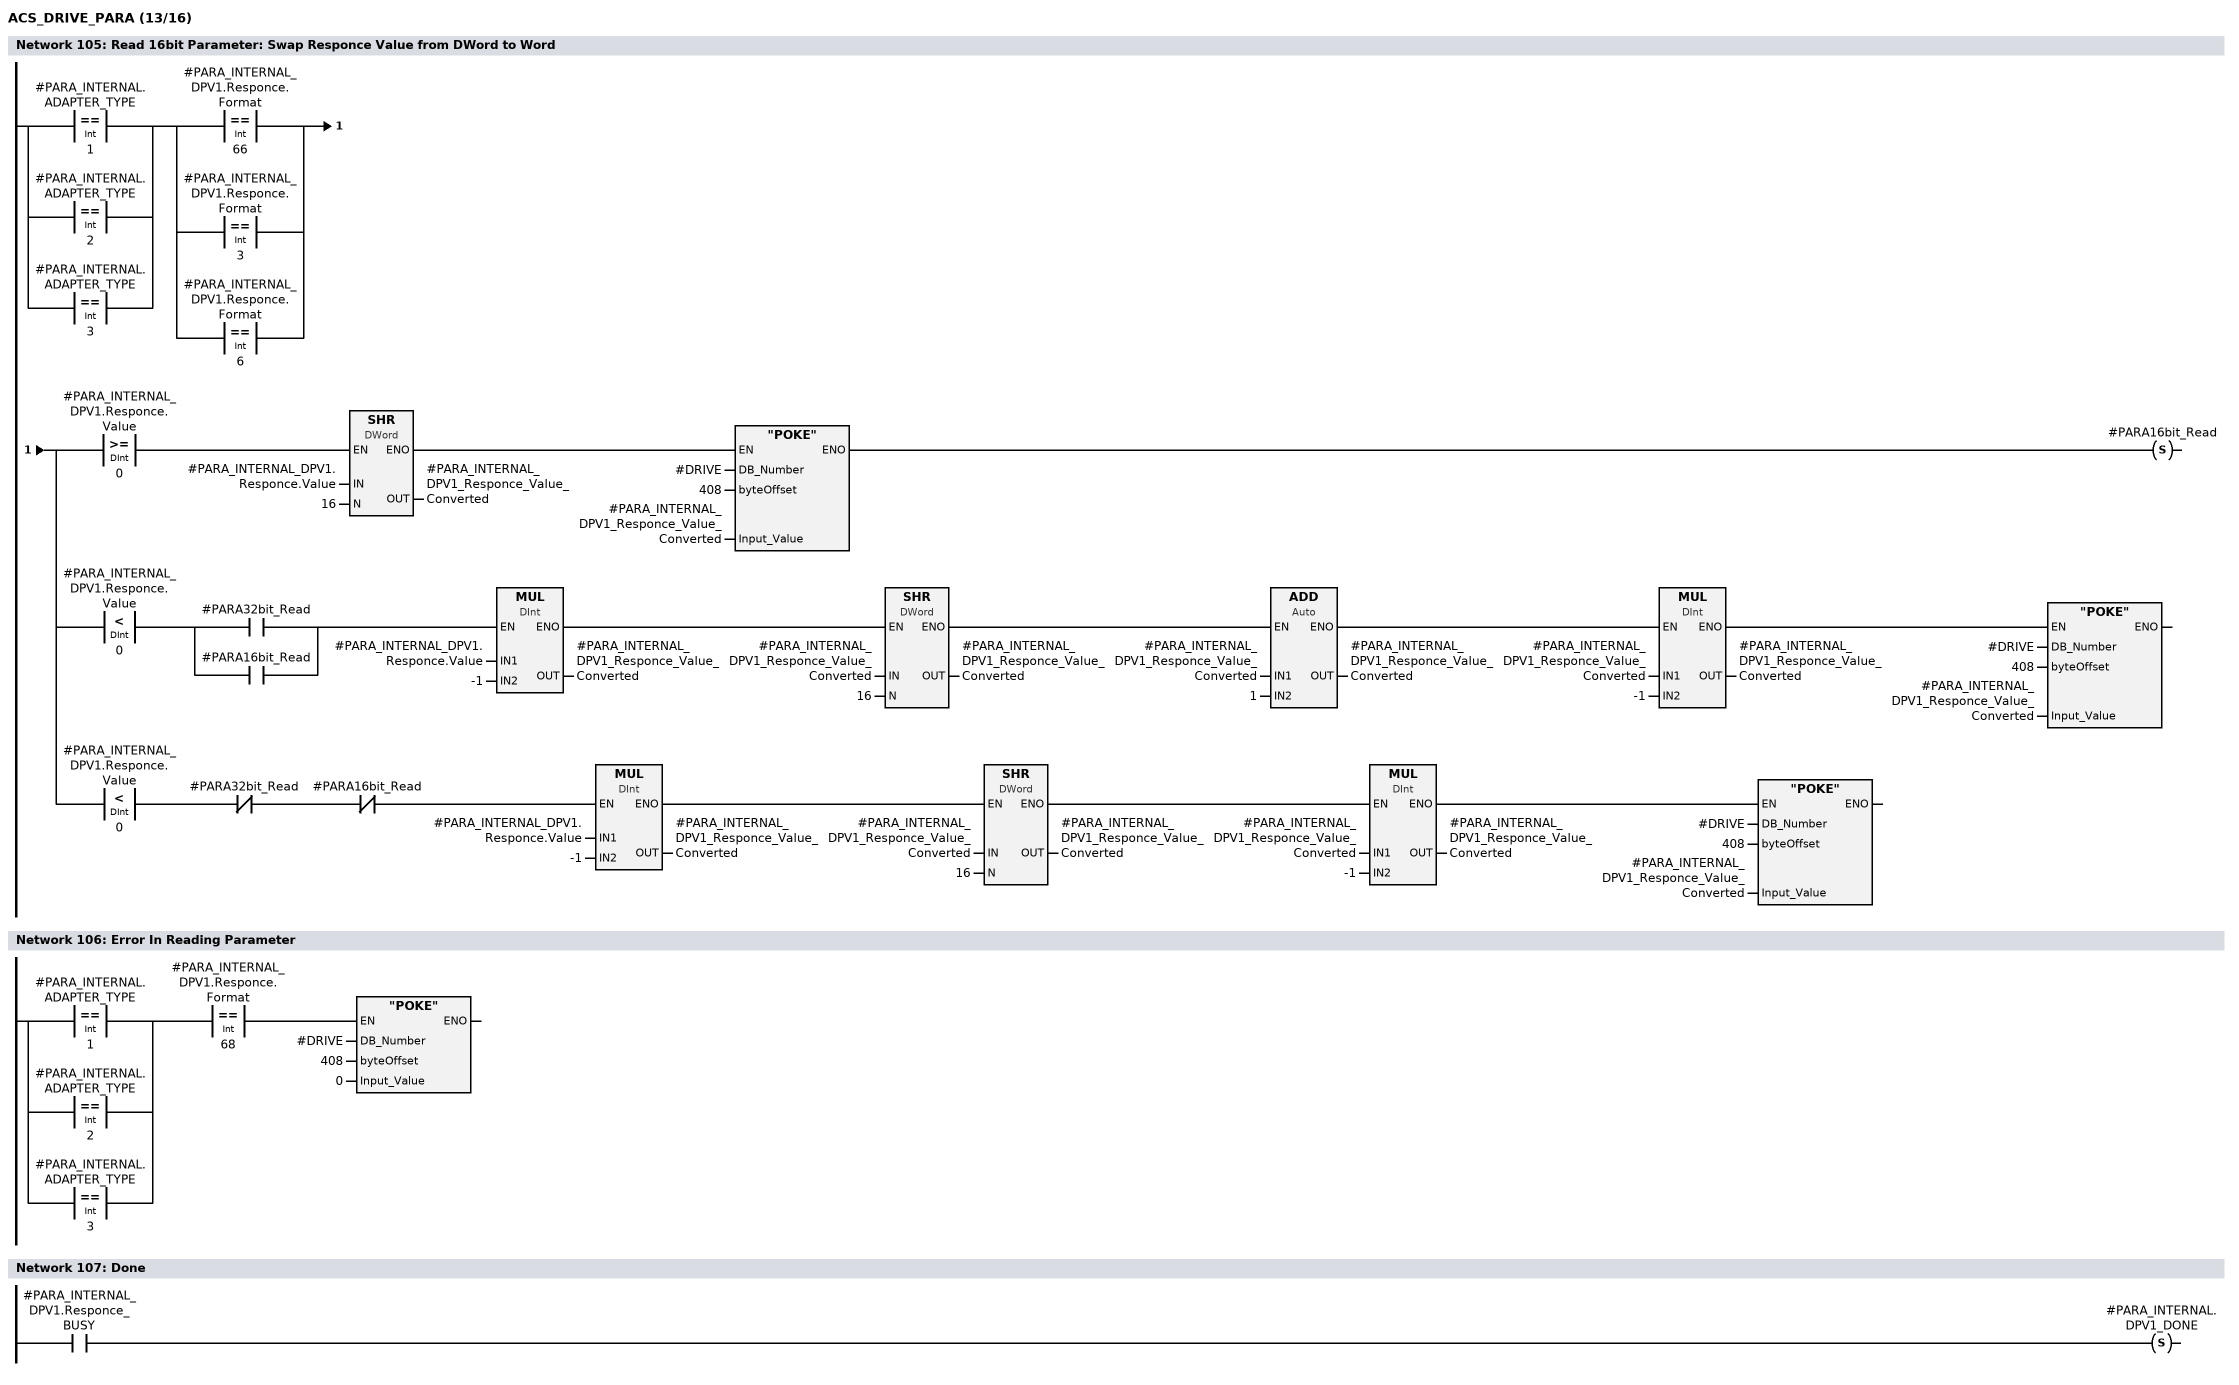
   RUNG wire#powerrail
      { S7_Templates := "SrcType := Int" } EQ_Contact(in1 := #PARA_INTERNAL.ADAPTER_TYPE, in2 := 1)
      wire#w1
      { S7_Templates := "SrcType := Int" } EQ_Contact(in1 := #PARA_INTERNAL_DPV1.Responce.Format, in2 := 66)
      wire#w2
      { S7_Templates := "SrcType := DInt" } GE_Contact(in1 := #PARA_INTERNAL_DPV1.Responce.Value, in2 := 0)
      { S7_Templates := "SrcType := DWord"; S7_GenerateENO := "TRUE" } Shr(in := #PARA_INTERNAL_DPV1.Responce.Value, n := 16, out => #PARA_INTERNAL_DPV1_Responce_Value_Converted)
      "POKE"(DB_Number := #DRIVE, byteOffset := 408, Input_Value := #PARA_INTERNAL_DPV1_Responce_Value_Converted)
      S_Coil( #PARA16bit_Read )
   END_RUNG
   RUNG wire#powerrail
      { S7_Templates := "SrcType := Int" } EQ_Contact(in1 := #PARA_INTERNAL.ADAPTER_TYPE, in2 := 2)
   END_RUNG wire#w1
   RUNG wire#powerrail
      { S7_Templates := "SrcType := Int" } EQ_Contact(in1 := #PARA_INTERNAL.ADAPTER_TYPE, in2 := 3)
   END_RUNG wire#w1
   RUNG wire#w1
      { S7_Templates := "SrcType := Int" } EQ_Contact(in1 := #PARA_INTERNAL_DPV1.Responce.Format, in2 := 3)
   END_RUNG wire#w2
   RUNG wire#w1
      { S7_Templates := "SrcType := Int" } EQ_Contact(in1 := #PARA_INTERNAL_DPV1.Responce.Format, in2 := 6)
   END_RUNG wire#w2
   RUNG wire#w2
      { S7_Templates := "SrcType := DInt" } LT_Contact(in1 := #PARA_INTERNAL_DPV1.Responce.Value, in2 := 0)
      wire#w3
      Contact( #PARA32bit_Read )
      wire#w4
      { S7_Templates := "SrcType := DInt" } Mul(in1 := #PARA_INTERNAL_DPV1.Responce.Value, in2 := -1, out => #PARA_INTERNAL_DPV1_Responce_Value_Converted)
      { S7_Templates := "SrcType := DWord"; S7_GenerateENO := "TRUE" } Shr(in := #PARA_INTERNAL_DPV1_Responce_Value_Converted, n := 16, out => #PARA_INTERNAL_DPV1_Responce_Value_Converted)
      Add(in1 := #PARA_INTERNAL_DPV1_Responce_Value_Converted, in2 := 1, out => #PARA_INTERNAL_DPV1_Responce_Value_Converted)
      { S7_Templates := "SrcType := DInt" } Mul(in1 := #PARA_INTERNAL_DPV1_Responce_Value_Converted, in2 := -1, out => #PARA_INTERNAL_DPV1_Responce_Value_Converted)
      "POKE"(DB_Number := #DRIVE, byteOffset := 408, Input_Value := #PARA_INTERNAL_DPV1_Responce_Value_Converted)
   END_RUNG
   RUNG wire#w3
      Contact( #PARA16bit_Read )
   END_RUNG wire#w4
   RUNG wire#w2
      { S7_Templates := "SrcType := DInt" } LT_Contact(in1 := #PARA_INTERNAL_DPV1.Responce.Value, in2 := 0)
      I_Contact( #PARA32bit_Read )
      I_Contact( #PARA16bit_Read )
      { S7_Templates := "SrcType := DInt" } Mul(in1 := #PARA_INTERNAL_DPV1.Responce.Value, in2 := -1, out => #PARA_INTERNAL_DPV1_Responce_Value_Converted)
      { S7_Templates := "SrcType := DWord"; S7_GenerateENO := "TRUE" } Shr(in := #PARA_INTERNAL_DPV1_Responce_Value_Converted, n := 16, out => #PARA_INTERNAL_DPV1_Responce_Value_Converted)
      { S7_Templates := "SrcType := DInt" } Mul(in1 := #PARA_INTERNAL_DPV1_Responce_Value_Converted, in2 := -1, out => #PARA_INTERNAL_DPV1_Responce_Value_Converted)
      "POKE"(DB_Number := #DRIVE, byteOffset := 408, Input_Value := #PARA_INTERNAL_DPV1_Responce_Value_Converted)
   END_RUNG
   // the same network as SCL:
   // ENO of a box is taken as its EN; it also drops when the box reports an error
   #_w1 := ((#PARA_INTERNAL.ADAPTER_TYPE = 1) OR (#PARA_INTERNAL.ADAPTER_TYPE = 2) OR (#PARA_INTERNAL.ADAPTER_TYPE = 3)) AND ((#PARA_INTERNAL_DPV1.Responce.Format = 66) OR (#PARA_INTERNAL_DPV1.Responce.Format = 3) OR (#PARA_INTERNAL_DPV1.Responce.Format = 6));
   IF #_w1 AND (#PARA_INTERNAL_DPV1.Responce.Value >= 0) THEN
       #PARA_INTERNAL_DPV1_Responce_Value_Converted := SHR(IN := #PARA_INTERNAL_DPV1.Responce.Value, N := 16);
   END_IF;
   "POKE"(EN := #_w1 AND (#PARA_INTERNAL_DPV1.Responce.Value >= 0),
          DB_Number := #DRIVE,
          byteOffset := 408,
          Input_Value := #PARA_INTERNAL_DPV1_Responce_Value_Converted,
          ENO => #_w2);
   IF #_w2 THEN #PARA16bit_Read := TRUE; END_IF;
   IF #_w1 AND (#PARA_INTERNAL_DPV1.Responce.Value < 0) AND (#PARA32bit_Read OR #PARA16bit_Read) THEN
       #PARA_INTERNAL_DPV1_Responce_Value_Converted := #PARA_INTERNAL_DPV1.Responce.Value * (-1);
       #PARA_INTERNAL_DPV1_Responce_Value_Converted := SHR(IN := #PARA_INTERNAL_DPV1_Responce_Value_Converted, N := 16);
       #PARA_INTERNAL_DPV1_Responce_Value_Converted := #PARA_INTERNAL_DPV1_Responce_Value_Converted + 1;
       #PARA_INTERNAL_DPV1_Responce_Value_Converted := #PARA_INTERNAL_DPV1_Responce_Value_Converted * (-1);
       "POKE"(DB_Number := #DRIVE, byteOffset := 408, Input_Value := #PARA_INTERNAL_DPV1_Responce_Value_Converted);
   END_IF;
   IF #_w1 AND (#PARA_INTERNAL_DPV1.Responce.Value < 0) AND NOT #PARA32bit_Read AND NOT #PARA16bit_Read THEN
       #PARA_INTERNAL_DPV1_Responce_Value_Converted := #PARA_INTERNAL_DPV1.Responce.Value * (-1);
       #PARA_INTERNAL_DPV1_Responce_Value_Converted := SHR(IN := #PARA_INTERNAL_DPV1_Responce_Value_Converted, N := 16);
       #PARA_INTERNAL_DPV1_Responce_Value_Converted := #PARA_INTERNAL_DPV1_Responce_Value_Converted * (-1);
       "POKE"(DB_Number := #DRIVE, byteOffset := 408, Input_Value := #PARA_INTERNAL_DPV1_Responce_Value_Converted);
   END_IF;
END_REGION

REGION Network 106: Error In Reading Parameter
   RUNG wire#powerrail
      { S7_Templates := "SrcType := Int" } EQ_Contact(in1 := #PARA_INTERNAL.ADAPTER_TYPE, in2 := 1)
      wire#w1
      { S7_Templates := "SrcType := Int" } EQ_Contact(in1 := #PARA_INTERNAL_DPV1.Responce.Format, in2 := 68)
      "POKE"(DB_Number := #DRIVE, byteOffset := 408, Input_Value := 0)
   END_RUNG
   RUNG wire#powerrail
      { S7_Templates := "SrcType := Int" } EQ_Contact(in1 := #PARA_INTERNAL.ADAPTER_TYPE, in2 := 2)
   END_RUNG wire#w1
   RUNG wire#powerrail
      { S7_Templates := "SrcType := Int" } EQ_Contact(in1 := #PARA_INTERNAL.ADAPTER_TYPE, in2 := 3)
   END_RUNG wire#w1
   // the same network as SCL:
   IF ((#PARA_INTERNAL.ADAPTER_TYPE = 1) OR (#PARA_INTERNAL.ADAPTER_TYPE = 2) OR (#PARA_INTERNAL.ADAPTER_TYPE = 3)) AND (#PARA_INTERNAL_DPV1.Responce.Format = 68) THEN
       "POKE"(DB_Number := #DRIVE, byteOffset := 408, Input_Value := 0);
   END_IF;
END_REGION

REGION Network 107: Done
   RUNG wire#powerrail
      Contact( #PARA_INTERNAL_DPV1.Responce_BUSY )
      S_Coil( #PARA_INTERNAL.DPV1_DONE )
   END_RUNG
   // the same network as SCL:
   IF #PARA_INTERNAL_DPV1.Responce_BUSY THEN #PARA_INTERNAL.DPV1_DONE := TRUE; END_IF;
END_REGION

REGION Network 108
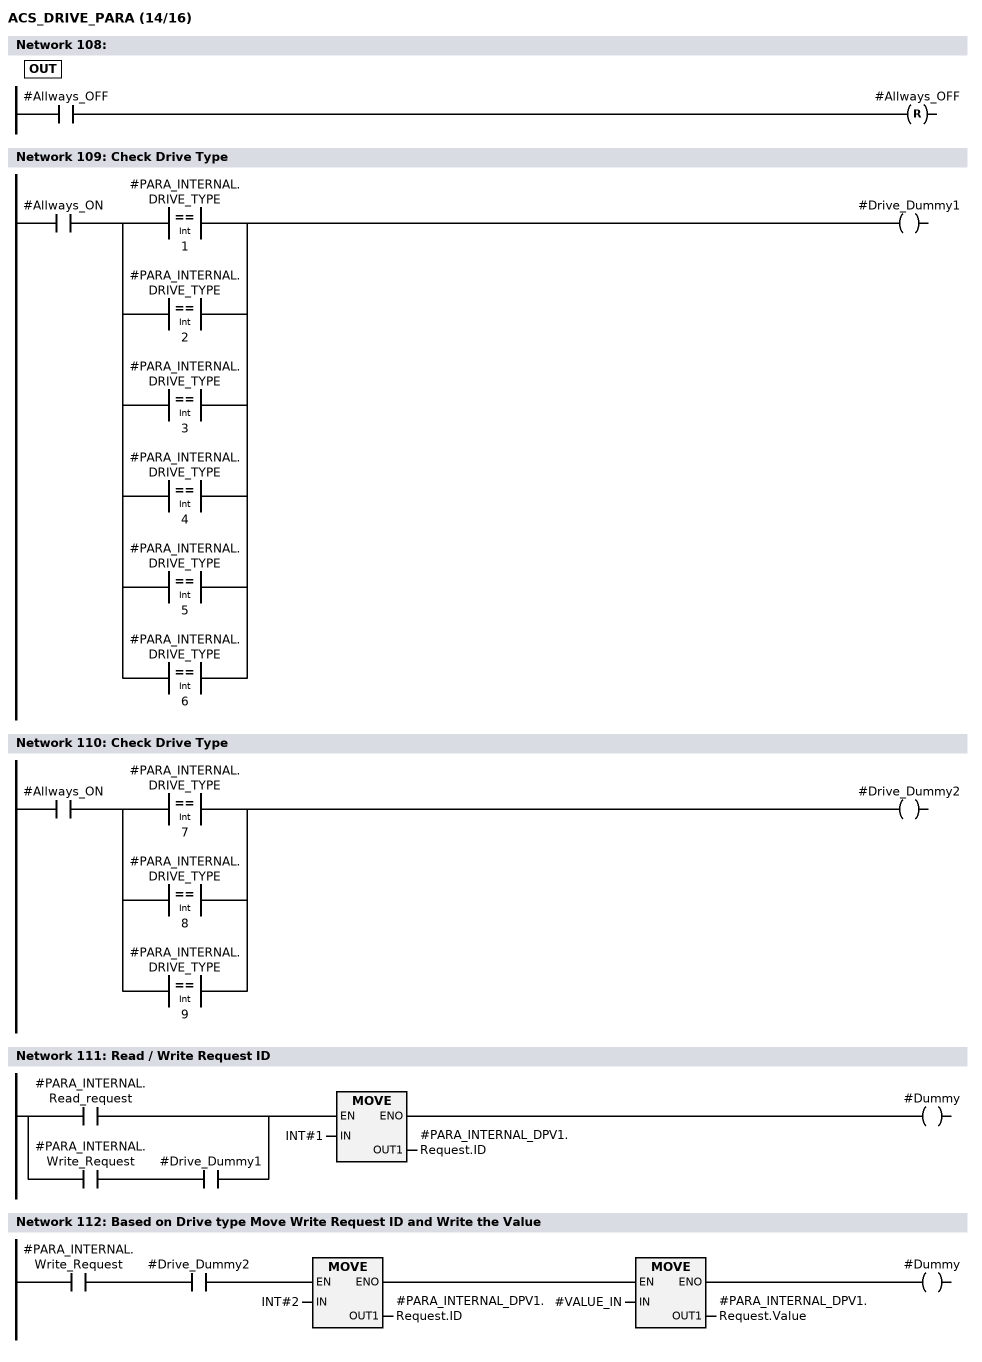
   Label( OUT )
   RUNG wire#powerrail
      Contact( #Allways_OFF )
      R_Coil( #Allways_OFF )
   END_RUNG
   // the same network as SCL:
   OUT:
   IF #Allways_OFF THEN #Allways_OFF := FALSE; END_IF;
END_REGION

REGION Network 109: Check Drive Type
   RUNG wire#powerrail
      Contact( #Allways_ON )
      wire#w1
      { S7_Templates := "SrcType := Int" } EQ_Contact(in1 := #PARA_INTERNAL.DRIVE_TYPE, in2 := 1)
      wire#w2
      Coil( #Drive_Dummy1 )
   END_RUNG
   RUNG wire#w1
      { S7_Templates := "SrcType := Int" } EQ_Contact(in1 := #PARA_INTERNAL.DRIVE_TYPE, in2 := 2)
   END_RUNG wire#w2
   RUNG wire#w1
      { S7_Templates := "SrcType := Int" } EQ_Contact(in1 := #PARA_INTERNAL.DRIVE_TYPE, in2 := 3)
   END_RUNG wire#w2
   RUNG wire#w1
      { S7_Templates := "SrcType := Int" } EQ_Contact(in1 := #PARA_INTERNAL.DRIVE_TYPE, in2 := 4)
   END_RUNG wire#w2
   RUNG wire#w1
      { S7_Templates := "SrcType := Int" } EQ_Contact(in1 := #PARA_INTERNAL.DRIVE_TYPE, in2 := 5)
   END_RUNG wire#w2
   RUNG wire#w1
      { S7_Templates := "SrcType := Int" } EQ_Contact(in1 := #PARA_INTERNAL.DRIVE_TYPE, in2 := 6)
   END_RUNG wire#w2
   // the same network as SCL:
   #Drive_Dummy1 := #Allways_ON AND ((#PARA_INTERNAL.DRIVE_TYPE = 1) OR (#PARA_INTERNAL.DRIVE_TYPE = 2) OR (#PARA_INTERNAL.DRIVE_TYPE = 3) OR (#PARA_INTERNAL.DRIVE_TYPE = 4) OR (#PARA_INTERNAL.DRIVE_TYPE = 5) OR (#PARA_INTERNAL.DRIVE_TYPE = 6));
END_REGION

REGION Network 110: Check Drive Type
   RUNG wire#powerrail
      Contact( #Allways_ON )
      wire#w1
      { S7_Templates := "SrcType := Int" } EQ_Contact(in1 := #PARA_INTERNAL.DRIVE_TYPE, in2 := 7)
      wire#w2
      Coil( #Drive_Dummy2 )
   END_RUNG
   RUNG wire#w1
      { S7_Templates := "SrcType := Int" } EQ_Contact(in1 := #PARA_INTERNAL.DRIVE_TYPE, in2 := 8)
   END_RUNG wire#w2
   RUNG wire#w1
      { S7_Templates := "SrcType := Int" } EQ_Contact(in1 := #PARA_INTERNAL.DRIVE_TYPE, in2 := 9)
   END_RUNG wire#w2
   // the same network as SCL:
   #Drive_Dummy2 := #Allways_ON AND ((#PARA_INTERNAL.DRIVE_TYPE = 7) OR (#PARA_INTERNAL.DRIVE_TYPE = 8) OR (#PARA_INTERNAL.DRIVE_TYPE = 9));
END_REGION

REGION Network 111: Read / Write Request ID
   RUNG wire#powerrail
      Contact( #PARA_INTERNAL.Read_request )
      wire#w1
      { S7_GenerateENO := "TRUE" } Move(in := INT#1, out1 => #PARA_INTERNAL_DPV1.Request.ID)
      Coil( #Dummy )
   END_RUNG
   RUNG wire#powerrail
      Contact( #PARA_INTERNAL.Write_Request )
      Contact( #Drive_Dummy1 )
   END_RUNG wire#w1
   // the same network as SCL:
   // ENO of a box is taken as its EN; it also drops when the box reports an error
   #_w1 := #PARA_INTERNAL.Read_request OR (#PARA_INTERNAL.Write_Request AND #Drive_Dummy1);
   IF #_w1 THEN #PARA_INTERNAL_DPV1.Request.ID := INT#1; END_IF;
   #Dummy := #_w1;
END_REGION

REGION Network 112: Based on Drive type Move Write Request ID and Write the Value
   RUNG wire#powerrail
      Contact( #PARA_INTERNAL.Write_Request )
      Contact( #Drive_Dummy2 )
      { S7_GenerateENO := "TRUE" } Move(in := INT#2, out1 => #PARA_INTERNAL_DPV1.Request.ID)
      { S7_GenerateENO := "TRUE" } Move(in := #VALUE_IN, out1 => #PARA_INTERNAL_DPV1.Request.Value)
      Coil( #Dummy )
   END_RUNG
   // the same network as SCL:
   // ENO of a box is taken as its EN; it also drops when the box reports an error
   #_w1 := #PARA_INTERNAL.Write_Request AND #Drive_Dummy2;
   IF #_w1 THEN
       #PARA_INTERNAL_DPV1.Request.ID := INT#2;
       #PARA_INTERNAL_DPV1.Request.Value := #VALUE_IN;
   END_IF;
   #Dummy := #_w1;
END_REGION

REGION Network 113: Based on Drive type Move Write Request ID & Write 16bit para val
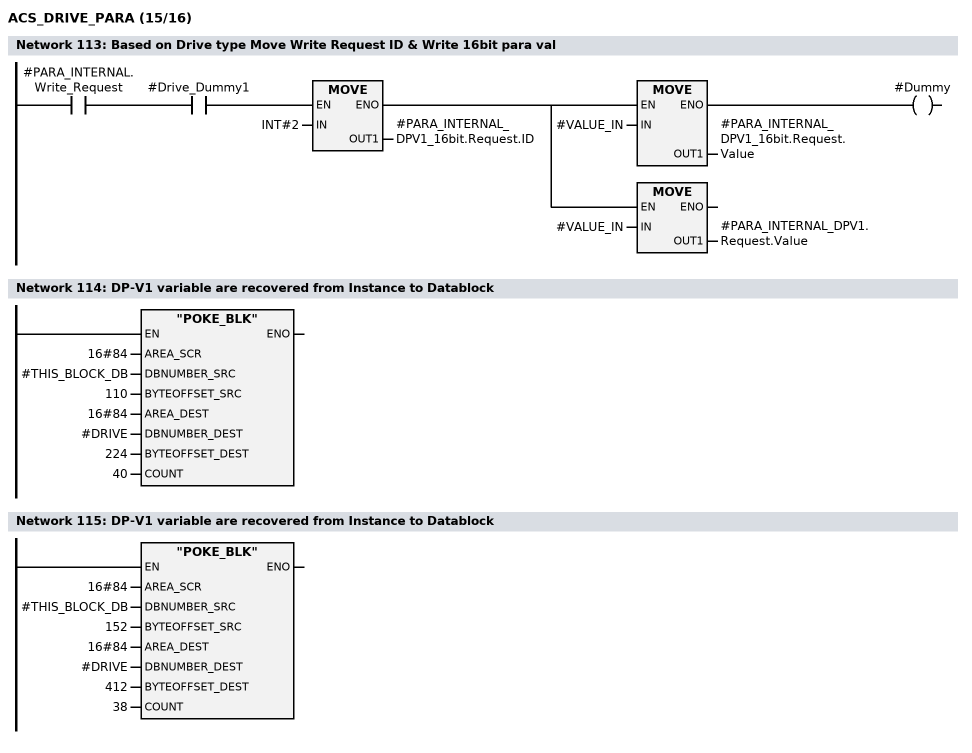
   RUNG wire#powerrail
      Contact( #PARA_INTERNAL.Write_Request )
      Contact( #Drive_Dummy1 )
      { S7_GenerateENO := "TRUE" } Move(in := INT#2, out1 => #PARA_INTERNAL_DPV1_16bit.Request.ID)
      wire#w1
      { S7_GenerateENO := "TRUE" } Move(in := #VALUE_IN, out1 => #PARA_INTERNAL_DPV1_16bit.Request.Value)
      Coil( #Dummy )
   END_RUNG
   RUNG wire#w1
      { S7_GenerateENO := "TRUE" } Move(in := #VALUE_IN, out1 => #PARA_INTERNAL_DPV1.Request.Value)
   END_RUNG
   // the same network as SCL:
   // ENO of a box is taken as its EN; it also drops when the box reports an error
   #_w1 := #PARA_INTERNAL.Write_Request AND #Drive_Dummy1;
   IF #_w1 THEN
       #PARA_INTERNAL_DPV1_16bit.Request.ID := INT#2;
       #PARA_INTERNAL_DPV1_16bit.Request.Value := #VALUE_IN;
   END_IF;
   #Dummy := #_w1;
   IF #_w1 THEN #PARA_INTERNAL_DPV1.Request.Value := #VALUE_IN; END_IF;
END_REGION

REGION Network 114: DP-V1 variable are recovered from Instance to Datablock
   RUNG wire#powerrail
      "POKE_BLK"(AREA_SCR := 16#84, DBNUMBER_SRC := #THIS_BLOCK_DB, BYTEOFFSET_SRC := 110, AREA_DEST := 16#84, DBNUMBER_DEST := #DRIVE, BYTEOFFSET_DEST := 224, COUNT := 40)
   END_RUNG
   // the same network as SCL:
   "POKE_BLK"(AREA_SCR := 16#84,
              DBNUMBER_SRC := #THIS_BLOCK_DB,
              BYTEOFFSET_SRC := 110,
              AREA_DEST := 16#84,
              DBNUMBER_DEST := #DRIVE,
              BYTEOFFSET_DEST := 224,
              COUNT := 40);
END_REGION

REGION Network 115: DP-V1 variable are recovered from Instance to Datablock
   RUNG wire#powerrail
      "POKE_BLK"(AREA_SCR := 16#84, DBNUMBER_SRC := #THIS_BLOCK_DB, BYTEOFFSET_SRC := 152, AREA_DEST := 16#84, DBNUMBER_DEST := #DRIVE, BYTEOFFSET_DEST := 412, COUNT := 38)
   END_RUNG
   // the same network as SCL:
   "POKE_BLK"(AREA_SCR := 16#84,
              DBNUMBER_SRC := #THIS_BLOCK_DB,
              BYTEOFFSET_SRC := 152,
              AREA_DEST := 16#84,
              DBNUMBER_DEST := #DRIVE,
              BYTEOFFSET_DEST := 412,
              COUNT := 38);
END_REGION

REGION Network 116: Output visualization
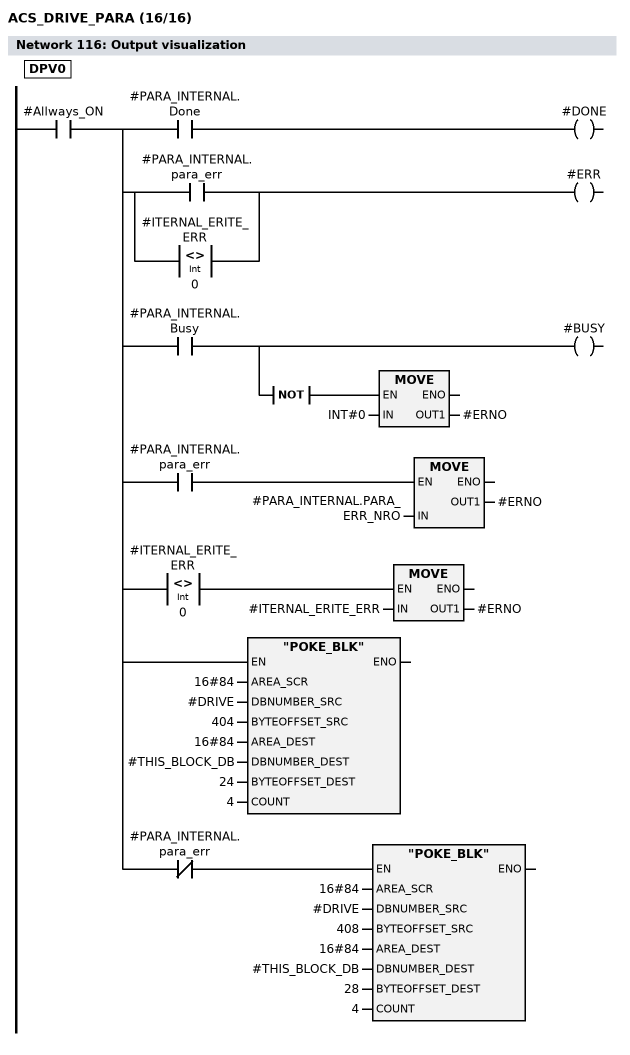
   Label( DPV0 )
   RUNG wire#powerrail
      Contact( #Allways_ON )
      wire#w1
      Contact( #PARA_INTERNAL.Done )
      Coil( #DONE )
   END_RUNG
   RUNG wire#w1
      Contact( #PARA_INTERNAL.para_err )
      wire#w2
      Coil( #ERR )
   END_RUNG
   RUNG wire#w1
      { S7_Templates := "SrcType := Int" } NE_Contact(in1 := #ITERNAL_ERITE_ERR, in2 := 0)
   END_RUNG wire#w2
   RUNG wire#w1
      Contact( #PARA_INTERNAL.Busy )
      wire#w3
      Coil( #BUSY )
   END_RUNG
   RUNG wire#w3
      Not()
      { S7_GenerateENO := "TRUE" } Move(in := INT#0, out1 => #ERNO)
   END_RUNG
   RUNG wire#w1
      Contact( #PARA_INTERNAL.para_err )
      { S7_GenerateENO := "TRUE" } Move(in := #PARA_INTERNAL.PARA_ERR_NRO, out1 => #ERNO)
   END_RUNG
   RUNG wire#w1
      { S7_Templates := "SrcType := Int" } NE_Contact(in1 := #ITERNAL_ERITE_ERR, in2 := 0)
      { S7_GenerateENO := "TRUE" } Move(in := #ITERNAL_ERITE_ERR, out1 => #ERNO)
   END_RUNG
   RUNG wire#w1
      "POKE_BLK"(AREA_SCR := 16#84, DBNUMBER_SRC := #DRIVE, BYTEOFFSET_SRC := 404, AREA_DEST := 16#84, DBNUMBER_DEST := #THIS_BLOCK_DB, BYTEOFFSET_DEST := 24, COUNT := 4)
   END_RUNG
   RUNG wire#w1
      I_Contact( #PARA_INTERNAL.para_err )
      "POKE_BLK"(AREA_SCR := 16#84, DBNUMBER_SRC := #DRIVE, BYTEOFFSET_SRC := 408, AREA_DEST := 16#84, DBNUMBER_DEST := #THIS_BLOCK_DB, BYTEOFFSET_DEST := 28, COUNT := 4)
   END_RUNG
   // the same network as SCL:
   DPV0:
   #DONE := #Allways_ON AND #PARA_INTERNAL.Done;
   #ERR := #Allways_ON AND (#PARA_INTERNAL.para_err OR (#ITERNAL_ERITE_ERR <> 0));
   #BUSY := #Allways_ON AND #PARA_INTERNAL.Busy;
   IF NOT #BUSY THEN #ERNO := INT#0; END_IF;
   IF #Allways_ON AND #PARA_INTERNAL.para_err THEN #ERNO := #PARA_INTERNAL.PARA_ERR_NRO; END_IF;
   IF #Allways_ON AND (#ITERNAL_ERITE_ERR <> 0) THEN #ERNO := #ITERNAL_ERITE_ERR; END_IF;
   IF #Allways_ON THEN
       "POKE_BLK"(AREA_SCR := 16#84,
                  DBNUMBER_SRC := #DRIVE,
                  BYTEOFFSET_SRC := 404,
                  AREA_DEST := 16#84,
                  DBNUMBER_DEST := #THIS_BLOCK_DB,
                  BYTEOFFSET_DEST := 24,
                  COUNT := 4);
   END_IF;
   IF #Allways_ON AND NOT #PARA_INTERNAL.para_err THEN
       "POKE_BLK"(AREA_SCR := 16#84,
                  DBNUMBER_SRC := #DRIVE,
                  BYTEOFFSET_SRC := 408,
                  AREA_DEST := 16#84,
                  DBNUMBER_DEST := #THIS_BLOCK_DB,
                  BYTEOFFSET_DEST := 28,
                  COUNT := 4);
   END_IF;
END_REGION
END_FUNCTION_BLOCK

FUNCTION_BLOCK "ACS_DRIVE_PZD"   // FB502, LAD
TITLE = ACS_DRIVE_PZD
{ S7_Optimized_Access := 'FALSE' }
AUTHOR : ABB
FAMILY : DRIVES
NAME : ABB
VERSION : 1.2
   VAR_INPUT
      PZD3_OUT : Int;   // Write PZD3 value to drive
      PZD4_OUT : Int;   // Write PZD4 value to drive
      PZD5_OUT : Int;   // Write PZD5 value to drive
      PZD6_OUT : Int;   // Write PZD6 value to drive
      PZD7_OUT : Int;   // Write PZD7 value to drive
      PZD8_OUT : Int;   // Write PZD8 value to drive
      PZD9_OUT : Int;   // Write PZD9 value to drive
      PZD10_OUT : Int;   // Write PZD10 value to drive
      Drive : DB_ANY;   // Instance DataBlock
      THIS_BLOCK_DB : DB_ANY;   // This Block instance DB
   END_VAR
   VAR_OUTPUT
      PZD2_SCALED : Real;   // Readed PZD2 scaled value
      PZD3_SCALED : Real;   // Readed PZD3 scaled value
      PZD4_SCALED : Real;   // Readed PZD4 scaled value
      PZD5_SCALED : Real;   // Readed PZD5 scaled value
      PZD6_SCALED : Real;   // Readed PZD6 scaled value
      PZD7_SCALED : Real;   // Readed PZD7 scaled value
      PZD8_SCALED : Real;   // Readed PZD8 scaled value
      PZD9_SCALED : Real;   // Readed PZD9 scaled value
      PZD10_SCALED : Real;   // Readed PZD10 scaled value
   END_VAR
   VAR
      ITERNAL_ERITE_ERR : Int;
      INTERNAL_PZD : Struct
         IN : Struct
            PZD2 : Int;   // 58
            PZD3 : Int;   // 60
            PZD4 : Int;   // 62
            PZD5 : Int;   // 64
            PZD6 : Int;   // 66
            PZD7 : Int;   // 68
            PZD8 : Int;   // 70
            PZD9 : Int;   // 72
            PZD10 : Int;   // 74
         END_STRUCT;
         OUT : Struct
            PZD3 : Int;   // 76
            PZD4 : Int;   // 78
            PZD5 : Int;   // 80
            PZD6 : Int;   // 82
            PZD7 : Int;   // 84
            PZD8 : Int;   // 86
            PZD9 : Int;   // 88
            PZD10 : Int;   // 90
         END_STRUCT;
         SCALED : Struct
            PZD2 : Real;   // 92
            PZD3 : Real;   // 96
            PZD4 : Real;   // 100
            PZD5 : Real;   // 104
            PZD6 : Real;   // 108
            PZD7 : Real;   // 112
            PZD8 : Real;   // 116
            PZD9 : Real;   // 120
            PZD10 : Real;   // 124
         END_STRUCT;
         SCALE : Struct
            PZD2_SCALE : Real;   // 128
            PZD3_SCALE : Real;   // 132
            PZD4_SCALE : Real;   // 136
            PZD5_SCALE : Real;   // 140
            PZD6_SCALE : Real;   // 144
            PZD7_SCALE : Real;   // 148
            PZD8_SCALE : Real;   // 152
            PZD9_SCALE : Real;   // 156
            PZD10_SCALE : Real;   // 160
         END_STRUCT;
      END_STRUCT;
      CONVERT_DI : DInt;
      CONVERTR_REAL : Real;
      PPO_TYPE : Int;   // PPO-Type: 1,2,3,4,5 or 6; 0 = no function
      NoPZD_Area : Bool;
      PPO_Type2_or_4_Selected : Bool;
   END_VAR
   VAR_TEMP
      Always_ON : Bool;
      Always_OFF : Bool;
   END_VAR
   VAR_TEMP   // added for the SCL form of the ladder/FBD networks
      _w1 : Bool;
      _w2 : Bool;
   END_VAR
BEGIN

REGION Network 1: Help flags
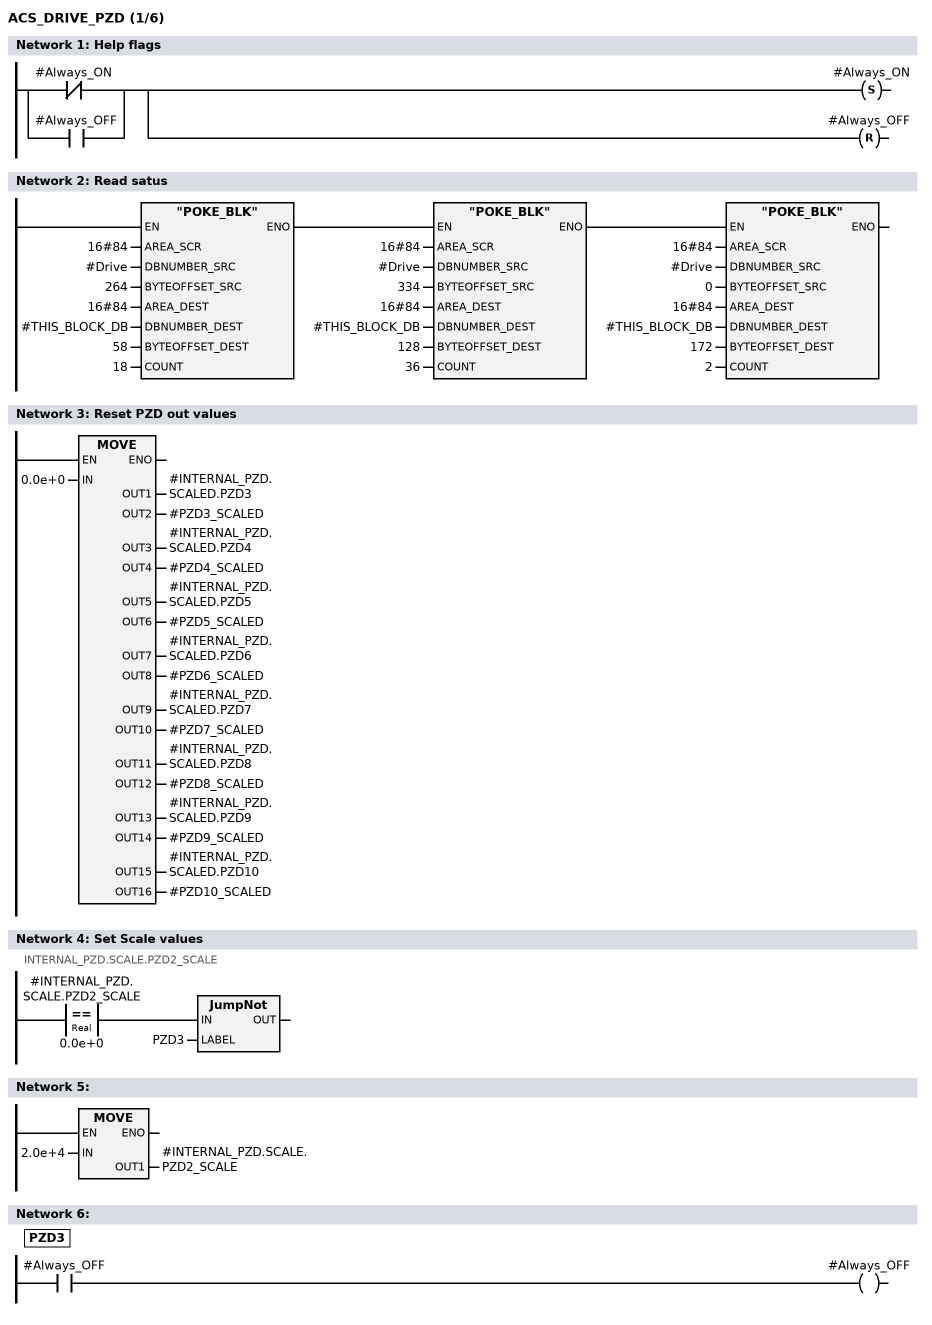
   RUNG wire#powerrail
      I_Contact( #Always_ON )
      wire#w1
      S_Coil( #Always_ON )
   END_RUNG
   RUNG wire#powerrail
      Contact( #Always_OFF )
   END_RUNG wire#w1
   RUNG wire#w1
      R_Coil( #Always_OFF )
   END_RUNG
   // the same network as SCL:
   #_w1 := NOT #Always_ON OR #Always_OFF;
   IF #_w1 THEN
       #Always_ON := TRUE;
       #Always_OFF := FALSE;
   END_IF;
END_REGION

REGION Network 2: Read satus
   RUNG wire#powerrail
      "POKE_BLK"(AREA_SCR := 16#84, DBNUMBER_SRC := #Drive, BYTEOFFSET_SRC := 264, AREA_DEST := 16#84, DBNUMBER_DEST := #THIS_BLOCK_DB, BYTEOFFSET_DEST := 58, COUNT := 18)
      "POKE_BLK"(AREA_SCR := 16#84, DBNUMBER_SRC := #Drive, BYTEOFFSET_SRC := 334, AREA_DEST := 16#84, DBNUMBER_DEST := #THIS_BLOCK_DB, BYTEOFFSET_DEST := 128, COUNT := 36)
      "POKE_BLK"(AREA_SCR := 16#84, DBNUMBER_SRC := #Drive, BYTEOFFSET_SRC := 0, AREA_DEST := 16#84, DBNUMBER_DEST := #THIS_BLOCK_DB, BYTEOFFSET_DEST := 172, COUNT := 2)
   END_RUNG
   // the same network as SCL:
   "POKE_BLK"(AREA_SCR := 16#84,
              DBNUMBER_SRC := #Drive,
              BYTEOFFSET_SRC := 264,
              AREA_DEST := 16#84,
              DBNUMBER_DEST := #THIS_BLOCK_DB,
              BYTEOFFSET_DEST := 58,
              COUNT := 18,
              ENO => #_w1);
   "POKE_BLK"(EN := #_w1,
              AREA_SCR := 16#84,
              DBNUMBER_SRC := #Drive,
              BYTEOFFSET_SRC := 334,
              AREA_DEST := 16#84,
              DBNUMBER_DEST := #THIS_BLOCK_DB,
              BYTEOFFSET_DEST := 128,
              COUNT := 36,
              ENO => #_w2);
   IF #_w2 THEN
       "POKE_BLK"(AREA_SCR := 16#84,
                  DBNUMBER_SRC := #Drive,
                  BYTEOFFSET_SRC := 0,
                  AREA_DEST := 16#84,
                  DBNUMBER_DEST := #THIS_BLOCK_DB,
                  BYTEOFFSET_DEST := 172,
                  COUNT := 2);
   END_IF;
END_REGION

REGION Network 3: Reset PZD out values
   RUNG wire#powerrail
      { S7_GenerateENO := "TRUE" } Move(in := 0.0e+0, out1 => #INTERNAL_PZD.SCALED.PZD3, out2 => #PZD3_SCALED, out3 => #INTERNAL_PZD.SCALED.PZD4, out4 => #PZD4_SCALED, out5 => #INTERNAL_PZD.SCALED.PZD5, out6 => #PZD5_SCALED, out7 => #INTERNAL_PZD.SCALED.PZD6, out8 => #PZD6_SCALED, out9 => #INTERNAL_PZD.SCALED.PZD7, out10 => #PZD7_SCALED, out11 => #INTERNAL_PZD.SCALED.PZD8, out12 => #PZD8_SCALED, out13 => #INTERNAL_PZD.SCALED.PZD9, out14 => #PZD9_SCALED, out15 => #INTERNAL_PZD.SCALED.PZD10, out16 => #PZD10_SCALED)
   END_RUNG
   // the same network as SCL:
   #INTERNAL_PZD.SCALED.PZD3 := 0.0e+0;
   #PZD3_SCALED := 0.0e+0;
   #INTERNAL_PZD.SCALED.PZD4 := 0.0e+0;
   #PZD4_SCALED := 0.0e+0;
   #INTERNAL_PZD.SCALED.PZD5 := 0.0e+0;
   #PZD5_SCALED := 0.0e+0;
   #INTERNAL_PZD.SCALED.PZD6 := 0.0e+0;
   #PZD6_SCALED := 0.0e+0;
   #INTERNAL_PZD.SCALED.PZD7 := 0.0e+0;
   #PZD7_SCALED := 0.0e+0;
   #INTERNAL_PZD.SCALED.PZD8 := 0.0e+0;
   #PZD8_SCALED := 0.0e+0;
   #INTERNAL_PZD.SCALED.PZD9 := 0.0e+0;
   #PZD9_SCALED := 0.0e+0;
   #INTERNAL_PZD.SCALED.PZD10 := 0.0e+0;
   #PZD10_SCALED := 0.0e+0;
END_REGION

REGION Network 4: Set Scale values
   // INTERNAL_PZD.SCALE.PZD2_SCALE
   // no SCL statement known for JumpNot: written as a call
   JumpNot(in := #INTERNAL_PZD.SCALE.PZD2_SCALE = 0.0e+0, label := PZD3);
END_REGION

REGION Network 5
   RUNG wire#powerrail
      { S7_GenerateENO := "TRUE" } Move(in := 2.0e+4, out1 => #INTERNAL_PZD.SCALE.PZD2_SCALE)
   END_RUNG
   // the same network as SCL:
   #INTERNAL_PZD.SCALE.PZD2_SCALE := 2.0e+4;
END_REGION

REGION Network 6
   Label( PZD3 )
   RUNG wire#powerrail
      Contact( #Always_OFF )
      Coil( #Always_OFF )
   END_RUNG
   // the same network as SCL:
   PZD3:
   #Always_OFF := #Always_OFF;
END_REGION

REGION Network 7
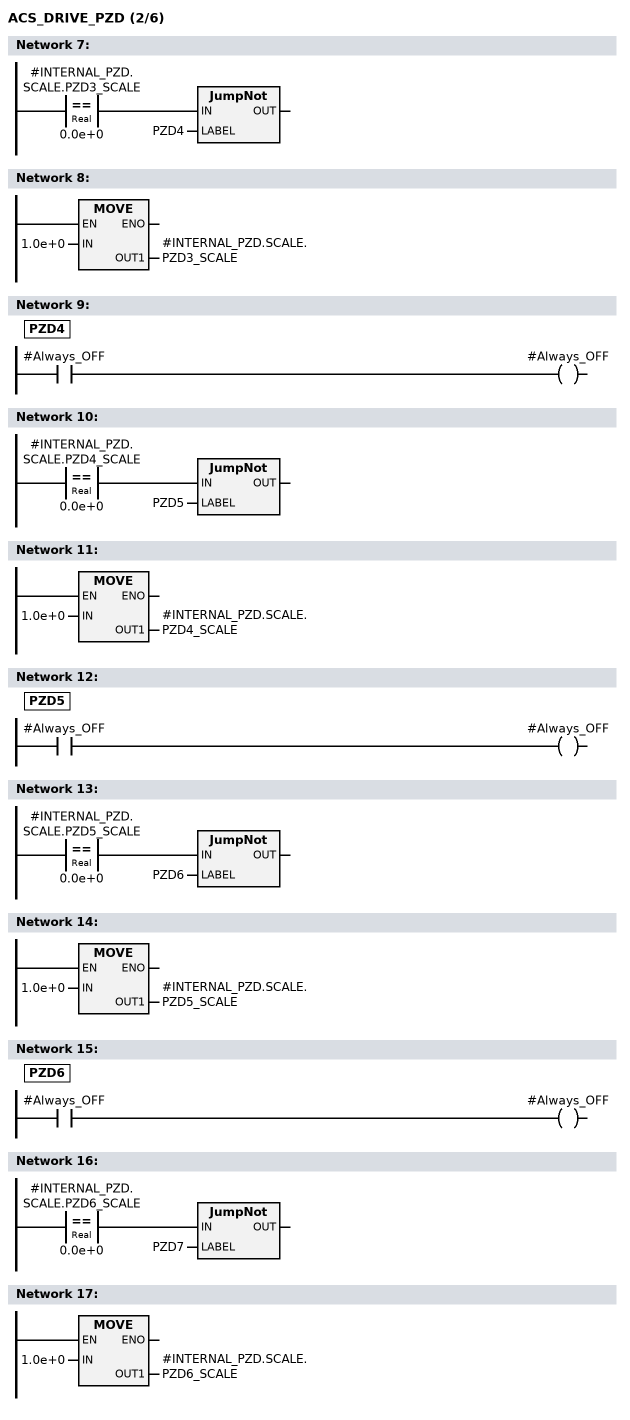
   // no SCL statement known for JumpNot: written as a call
   JumpNot(in := #INTERNAL_PZD.SCALE.PZD3_SCALE = 0.0e+0, label := PZD4);
END_REGION

REGION Network 8
   RUNG wire#powerrail
      { S7_GenerateENO := "TRUE" } Move(in := 1.0e+0, out1 => #INTERNAL_PZD.SCALE.PZD3_SCALE)
   END_RUNG
   // the same network as SCL:
   #INTERNAL_PZD.SCALE.PZD3_SCALE := 1.0e+0;
END_REGION

REGION Network 9
   Label( PZD4 )
   RUNG wire#powerrail
      Contact( #Always_OFF )
      Coil( #Always_OFF )
   END_RUNG
   // the same network as SCL:
   PZD4:
   #Always_OFF := #Always_OFF;
END_REGION

REGION Network 10
   // no SCL statement known for JumpNot: written as a call
   JumpNot(in := #INTERNAL_PZD.SCALE.PZD4_SCALE = 0.0e+0, label := PZD5);
END_REGION

REGION Network 11
   RUNG wire#powerrail
      { S7_GenerateENO := "TRUE" } Move(in := 1.0e+0, out1 => #INTERNAL_PZD.SCALE.PZD4_SCALE)
   END_RUNG
   // the same network as SCL:
   #INTERNAL_PZD.SCALE.PZD4_SCALE := 1.0e+0;
END_REGION

REGION Network 12
   Label( PZD5 )
   RUNG wire#powerrail
      Contact( #Always_OFF )
      Coil( #Always_OFF )
   END_RUNG
   // the same network as SCL:
   PZD5:
   #Always_OFF := #Always_OFF;
END_REGION

REGION Network 13
   // no SCL statement known for JumpNot: written as a call
   JumpNot(in := #INTERNAL_PZD.SCALE.PZD5_SCALE = 0.0e+0, label := PZD6);
END_REGION

REGION Network 14
   RUNG wire#powerrail
      { S7_GenerateENO := "TRUE" } Move(in := 1.0e+0, out1 => #INTERNAL_PZD.SCALE.PZD5_SCALE)
   END_RUNG
   // the same network as SCL:
   #INTERNAL_PZD.SCALE.PZD5_SCALE := 1.0e+0;
END_REGION

REGION Network 15
   Label( PZD6 )
   RUNG wire#powerrail
      Contact( #Always_OFF )
      Coil( #Always_OFF )
   END_RUNG
   // the same network as SCL:
   PZD6:
   #Always_OFF := #Always_OFF;
END_REGION

REGION Network 16
   // no SCL statement known for JumpNot: written as a call
   JumpNot(in := #INTERNAL_PZD.SCALE.PZD6_SCALE = 0.0e+0, label := PZD7);
END_REGION

REGION Network 17
   RUNG wire#powerrail
      { S7_GenerateENO := "TRUE" } Move(in := 1.0e+0, out1 => #INTERNAL_PZD.SCALE.PZD6_SCALE)
   END_RUNG
   // the same network as SCL:
   #INTERNAL_PZD.SCALE.PZD6_SCALE := 1.0e+0;
END_REGION

REGION Network 18
